REGION Network 96: Transfer P&P Left AxisX Home Interlock Condition
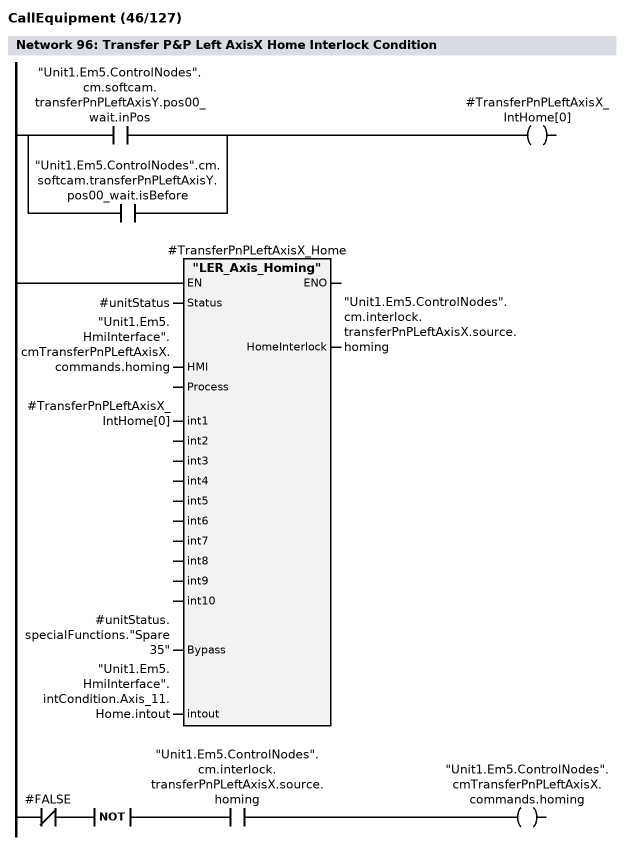
   RUNG wire#powerrail
      Contact( "Unit1.Em5.ControlNodes".cm.softcam.transferPnPLeftAxisY.pos00_wait.inPos )
      wire#w1
      Coil( #TransferPnPLeftAxisX_IntHome[0] )
   END_RUNG
   RUNG wire#powerrail
      Contact( "Unit1.Em5.ControlNodes".cm.softcam.transferPnPLeftAxisY.pos00_wait.isBefore )
   END_RUNG wire#w1
   RUNG wire#powerrail
      #TransferPnPLeftAxisX_Home(Status := #unitStatus, HMI := "Unit1.Em5.HmiInterface".cmTransferPnPLeftAxisX.commands.homing, Process :=, int1 := #TransferPnPLeftAxisX_IntHome[0], int2 :=, int3 :=, int4 :=, int5 :=, int6 :=, int7 :=, int8 :=, int9 :=, int10 :=, Bypass := #unitStatus.specialFunctions."Spare 35", intout := "Unit1.Em5.HmiInterface".intCondition.Axis_11.Home.intout, HomeInterlock => "Unit1.Em5.ControlNodes".cm.interlock.transferPnPLeftAxisX.source.homing)
   END_RUNG
   RUNG wire#powerrail
      I_Contact( #FALSE )
      Not()
      Contact( "Unit1.Em5.ControlNodes".cm.interlock.transferPnPLeftAxisX.source.homing )
      Coil( "Unit1.Em5.ControlNodes".cmTransferPnPLeftAxisX.commands.homing )
   END_RUNG
   // the same network as SCL:
   #TransferPnPLeftAxisX_IntHome[0] := "Unit1.Em5.ControlNodes".cm.softcam.transferPnPLeftAxisY.pos00_wait.inPos OR "Unit1.Em5.ControlNodes".cm.softcam.transferPnPLeftAxisY.pos00_wait.isBefore;
   #TransferPnPLeftAxisX_Home(Status := #unitStatus,   // "LER_Axis_Homing"
                           HMI := "Unit1.Em5.HmiInterface".cmTransferPnPLeftAxisX.commands.homing,
                           int1 := #TransferPnPLeftAxisX_IntHome[0],
                           Bypass := #unitStatus.specialFunctions."Spare 35",
                           intout := "Unit1.Em5.HmiInterface".intCondition.Axis_11.Home.intout,
                           HomeInterlock => "Unit1.Em5.ControlNodes".cm.interlock.transferPnPLeftAxisX.source.homing);
   "Unit1.Em5.ControlNodes".cmTransferPnPLeftAxisX.commands.homing := NOT (NOT #FALSE) AND "Unit1.Em5.ControlNodes".cm.interlock.transferPnPLeftAxisX.source.homing;
END_REGION

REGION Network 97: Transfer P&P Left AxisX JOG Interlock Condition
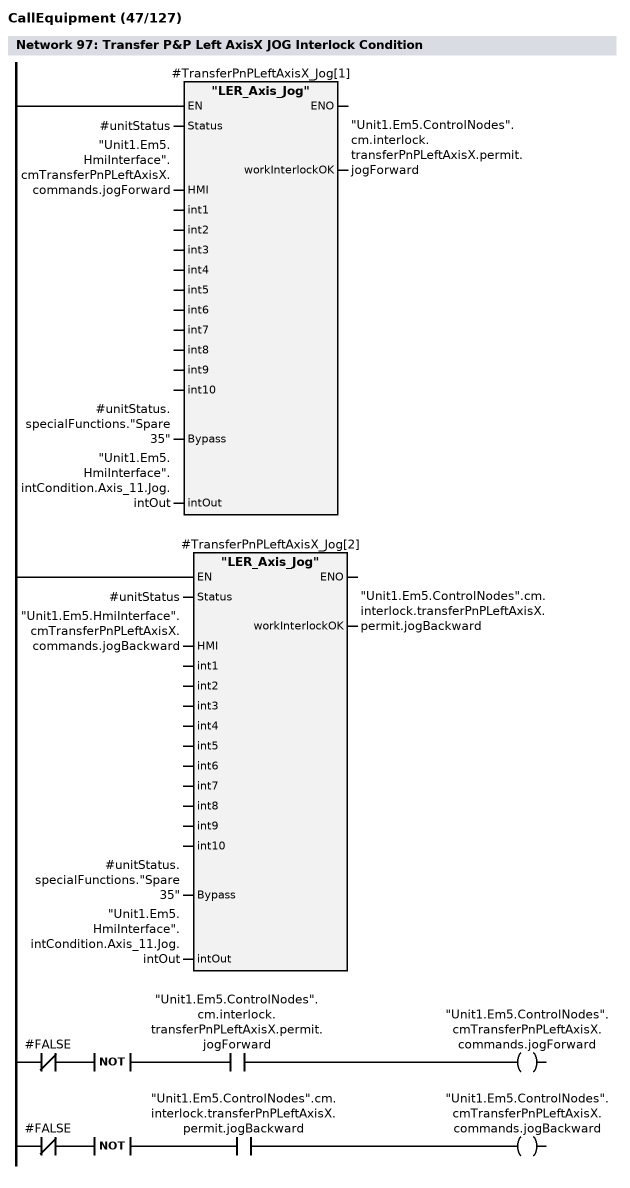
   RUNG wire#powerrail
      #TransferPnPLeftAxisX_Jog[1](Status := #unitStatus, HMI := "Unit1.Em5.HmiInterface".cmTransferPnPLeftAxisX.commands.jogForward, int1 :=, int2 :=, int3 :=, int4 :=, int5 :=, int6 :=, int7 :=, int8 :=, int9 :=, int10 :=, Bypass := #unitStatus.specialFunctions."Spare 35", intOut := "Unit1.Em5.HmiInterface".intCondition.Axis_11.Jog.intOut, workInterlockOK => "Unit1.Em5.ControlNodes".cm.interlock.transferPnPLeftAxisX.permit.jogForward)
   END_RUNG
   RUNG wire#powerrail
      #TransferPnPLeftAxisX_Jog[2](Status := #unitStatus, HMI := "Unit1.Em5.HmiInterface".cmTransferPnPLeftAxisX.commands.jogBackward, int1 :=, int2 :=, int3 :=, int4 :=, int5 :=, int6 :=, int7 :=, int8 :=, int9 :=, int10 :=, Bypass := #unitStatus.specialFunctions."Spare 35", intOut := "Unit1.Em5.HmiInterface".intCondition.Axis_11.Jog.intOut, workInterlockOK => "Unit1.Em5.ControlNodes".cm.interlock.transferPnPLeftAxisX.permit.jogBackward)
   END_RUNG
   RUNG wire#powerrail
      I_Contact( #FALSE )
      Not()
      Contact( "Unit1.Em5.ControlNodes".cm.interlock.transferPnPLeftAxisX.permit.jogForward )
      Coil( "Unit1.Em5.ControlNodes".cmTransferPnPLeftAxisX.commands.jogForward )
   END_RUNG
   RUNG wire#powerrail
      I_Contact( #FALSE )
      Not()
      Contact( "Unit1.Em5.ControlNodes".cm.interlock.transferPnPLeftAxisX.permit.jogBackward )
      Coil( "Unit1.Em5.ControlNodes".cmTransferPnPLeftAxisX.commands.jogBackward )
   END_RUNG
   // the same network as SCL:
   #TransferPnPLeftAxisX_Jog[1](Status := #unitStatus,   // "LER_Axis_Jog"
                           HMI := "Unit1.Em5.HmiInterface".cmTransferPnPLeftAxisX.commands.jogForward,
                           Bypass := #unitStatus.specialFunctions."Spare 35",
                           intOut := "Unit1.Em5.HmiInterface".intCondition.Axis_11.Jog.intOut,
                           workInterlockOK => "Unit1.Em5.ControlNodes".cm.interlock.transferPnPLeftAxisX.permit.jogForward);
   #TransferPnPLeftAxisX_Jog[2](Status := #unitStatus,   // "LER_Axis_Jog"
                           HMI := "Unit1.Em5.HmiInterface".cmTransferPnPLeftAxisX.commands.jogBackward,
                           Bypass := #unitStatus.specialFunctions."Spare 35",
                           intOut := "Unit1.Em5.HmiInterface".intCondition.Axis_11.Jog.intOut,
                           workInterlockOK => "Unit1.Em5.ControlNodes".cm.interlock.transferPnPLeftAxisX.permit.jogBackward);
   "Unit1.Em5.ControlNodes".cmTransferPnPLeftAxisX.commands.jogForward := NOT (NOT #FALSE) AND "Unit1.Em5.ControlNodes".cm.interlock.transferPnPLeftAxisX.permit.jogForward;
   "Unit1.Em5.ControlNodes".cmTransferPnPLeftAxisX.commands.jogBackward := NOT (NOT #FALSE) AND "Unit1.Em5.ControlNodes".cm.interlock.transferPnPLeftAxisX.permit.jogBackward;
END_REGION

REGION Network 98: Transfer P&P Left AxisX Position Absolute Position0
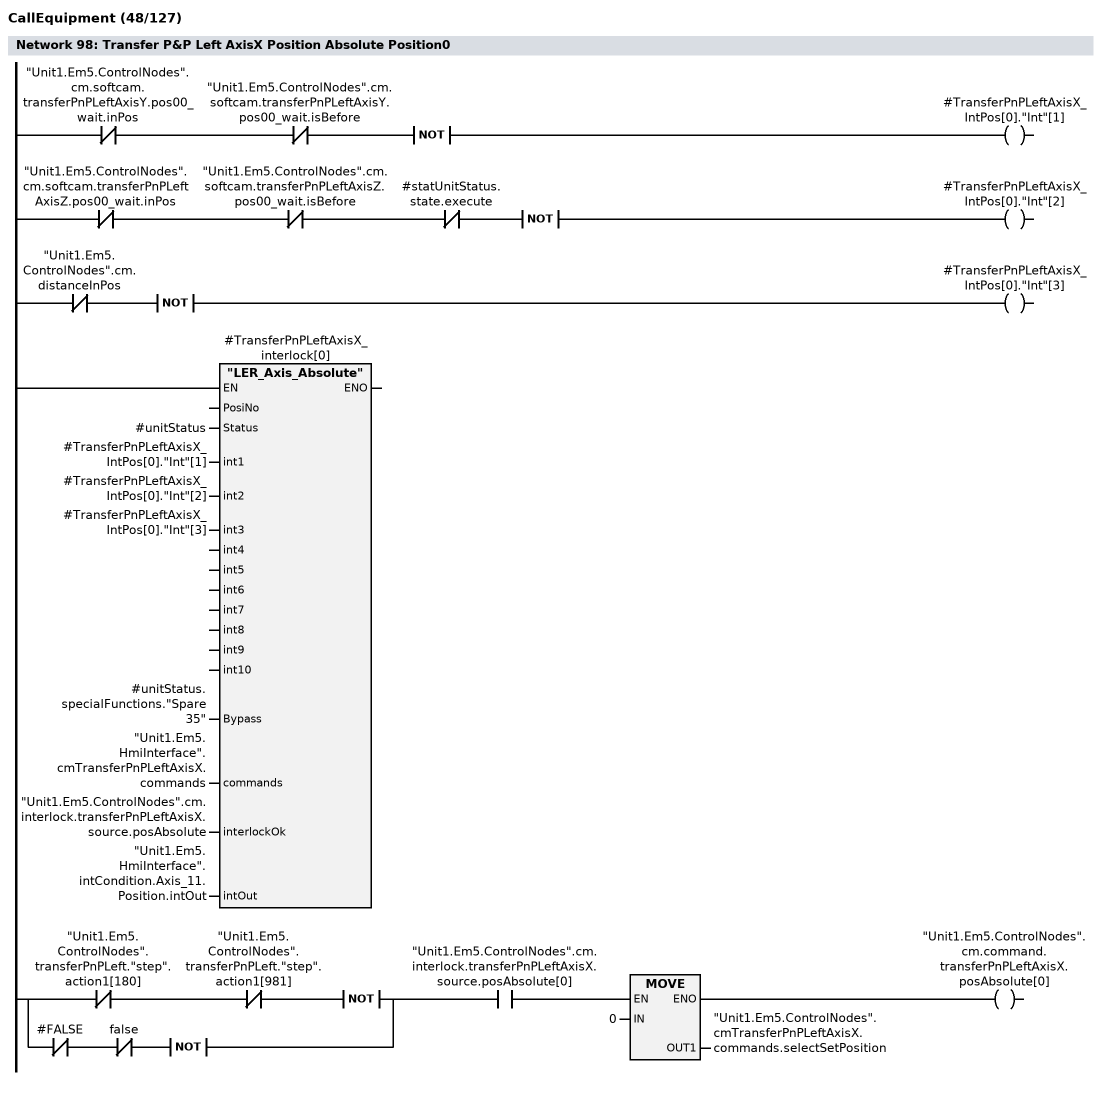
   RUNG wire#powerrail
      I_Contact( "Unit1.Em5.ControlNodes".cm.softcam.transferPnPLeftAxisY.pos00_wait.inPos )
      I_Contact( "Unit1.Em5.ControlNodes".cm.softcam.transferPnPLeftAxisY.pos00_wait.isBefore )
      Not()
      Coil( #TransferPnPLeftAxisX_IntPos[0]."Int"[1] )
   END_RUNG
   RUNG wire#powerrail
      I_Contact( "Unit1.Em5.ControlNodes".cm.softcam.transferPnPLeftAxisZ.pos00_wait.inPos )
      I_Contact( "Unit1.Em5.ControlNodes".cm.softcam.transferPnPLeftAxisZ.pos00_wait.isBefore )
      I_Contact( #statUnitStatus.state.execute )
      Not()
      Coil( #TransferPnPLeftAxisX_IntPos[0]."Int"[2] )
   END_RUNG
   RUNG wire#powerrail
      I_Contact( "Unit1.Em5.ControlNodes".cm.distanceInPos )
      Not()
      Coil( #TransferPnPLeftAxisX_IntPos[0]."Int"[3] )
   END_RUNG
   RUNG wire#powerrail
      #TransferPnPLeftAxisX_interlock[0](PosiNo :=, Status := #unitStatus, int1 := #TransferPnPLeftAxisX_IntPos[0]."Int"[1], int2 := #TransferPnPLeftAxisX_IntPos[0]."Int"[2], int3 := #TransferPnPLeftAxisX_IntPos[0]."Int"[3], int4 :=, int5 :=, int6 :=, int7 :=, int8 :=, int9 :=, int10 :=, Bypass := #unitStatus.specialFunctions."Spare 35", commands := "Unit1.Em5.HmiInterface".cmTransferPnPLeftAxisX.commands, interlockOk := "Unit1.Em5.ControlNodes".cm.interlock.transferPnPLeftAxisX.source.posAbsolute, intOut := "Unit1.Em5.HmiInterface".intCondition.Axis_11.Position.intOut)
   END_RUNG
   RUNG wire#powerrail
      I_Contact( "Unit1.Em5.ControlNodes".transferPnPLeft."step".action1[180] )
      I_Contact( "Unit1.Em5.ControlNodes".transferPnPLeft."step".action1[981] )
      Not()
      wire#w1
      Contact( "Unit1.Em5.ControlNodes".cm.interlock.transferPnPLeftAxisX.source.posAbsolute[0] )
      Move(in := 0, out1 => "Unit1.Em5.ControlNodes".cmTransferPnPLeftAxisX.commands.selectSetPosition)
      Coil( "Unit1.Em5.ControlNodes".cm.command.transferPnPLeftAxisX.posAbsolute[0] )
   END_RUNG
   RUNG wire#powerrail
      I_Contact( #FALSE )
      I_Contact( false )
      Not()
   END_RUNG wire#w1
   // the same network as SCL:
   #TransferPnPLeftAxisX_IntPos[0]."Int"[1] := NOT (NOT "Unit1.Em5.ControlNodes".cm.softcam.transferPnPLeftAxisY.pos00_wait.inPos AND NOT "Unit1.Em5.ControlNodes".cm.softcam.transferPnPLeftAxisY.pos00_wait.isBefore);
   #TransferPnPLeftAxisX_IntPos[0]."Int"[2] := NOT (NOT "Unit1.Em5.ControlNodes".cm.softcam.transferPnPLeftAxisZ.pos00_wait.inPos AND NOT "Unit1.Em5.ControlNodes".cm.softcam.transferPnPLeftAxisZ.pos00_wait.isBefore AND NOT #statUnitStatus.state.execute);
   #TransferPnPLeftAxisX_IntPos[0]."Int"[3] := NOT (NOT "Unit1.Em5.ControlNodes".cm.distanceInPos);
   #TransferPnPLeftAxisX_interlock[0](Status := #unitStatus,   // "LER_Axis_Absolute"
                           int1 := #TransferPnPLeftAxisX_IntPos[0]."Int"[1],
                           int2 := #TransferPnPLeftAxisX_IntPos[0]."Int"[2],
                           int3 := #TransferPnPLeftAxisX_IntPos[0]."Int"[3],
                           Bypass := #unitStatus.specialFunctions."Spare 35",
                           commands := "Unit1.Em5.HmiInterface".cmTransferPnPLeftAxisX.commands,
                           interlockOk := "Unit1.Em5.ControlNodes".cm.interlock.transferPnPLeftAxisX.source.posAbsolute,
                           intOut := "Unit1.Em5.HmiInterface".intCondition.Axis_11.Position.intOut);
   #_w1 := (NOT (NOT "Unit1.Em5.ControlNodes".transferPnPLeft."step".action1[180] AND NOT "Unit1.Em5.ControlNodes".transferPnPLeft."step".action1[981]) OR NOT (NOT #FALSE AND NOT false)) AND "Unit1.Em5.ControlNodes".cm.interlock.transferPnPLeftAxisX.source.posAbsolute[0];
   IF #_w1 THEN "Unit1.Em5.ControlNodes".cmTransferPnPLeftAxisX.commands.selectSetPosition := 0; END_IF;
   "Unit1.Em5.ControlNodes".cm.command.transferPnPLeftAxisX.posAbsolute[0] := #_w1;
END_REGION

REGION Network 99: Transfer P&P Left AxisX Position Absolute Position1
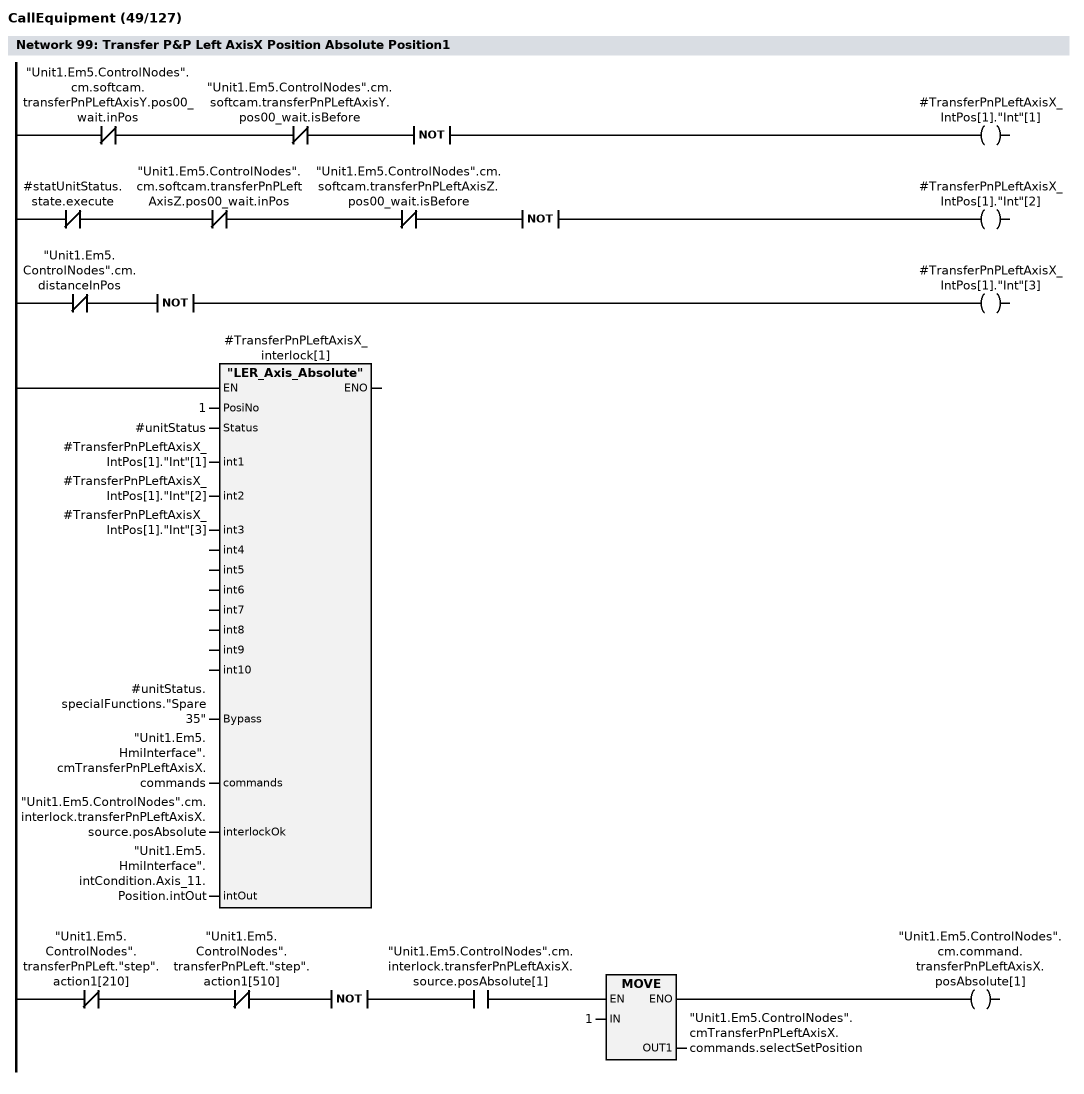
   RUNG wire#powerrail
      I_Contact( "Unit1.Em5.ControlNodes".cm.softcam.transferPnPLeftAxisY.pos00_wait.inPos )
      I_Contact( "Unit1.Em5.ControlNodes".cm.softcam.transferPnPLeftAxisY.pos00_wait.isBefore )
      Not()
      Coil( #TransferPnPLeftAxisX_IntPos[1]."Int"[1] )
   END_RUNG
   RUNG wire#powerrail
      I_Contact( #statUnitStatus.state.execute )
      I_Contact( "Unit1.Em5.ControlNodes".cm.softcam.transferPnPLeftAxisZ.pos00_wait.inPos )
      I_Contact( "Unit1.Em5.ControlNodes".cm.softcam.transferPnPLeftAxisZ.pos00_wait.isBefore )
      Not()
      Coil( #TransferPnPLeftAxisX_IntPos[1]."Int"[2] )
   END_RUNG
   RUNG wire#powerrail
      I_Contact( "Unit1.Em5.ControlNodes".cm.distanceInPos )
      Not()
      Coil( #TransferPnPLeftAxisX_IntPos[1]."Int"[3] )
   END_RUNG
   RUNG wire#powerrail
      #TransferPnPLeftAxisX_interlock[1](PosiNo := 1, Status := #unitStatus, int1 := #TransferPnPLeftAxisX_IntPos[1]."Int"[1], int2 := #TransferPnPLeftAxisX_IntPos[1]."Int"[2], int3 := #TransferPnPLeftAxisX_IntPos[1]."Int"[3], int4 :=, int5 :=, int6 :=, int7 :=, int8 :=, int9 :=, int10 :=, Bypass := #unitStatus.specialFunctions."Spare 35", commands := "Unit1.Em5.HmiInterface".cmTransferPnPLeftAxisX.commands, interlockOk := "Unit1.Em5.ControlNodes".cm.interlock.transferPnPLeftAxisX.source.posAbsolute, intOut := "Unit1.Em5.HmiInterface".intCondition.Axis_11.Position.intOut)
   END_RUNG
   RUNG wire#powerrail
      I_Contact( "Unit1.Em5.ControlNodes".transferPnPLeft."step".action1[210] )
      I_Contact( "Unit1.Em5.ControlNodes".transferPnPLeft."step".action1[510] )
      Not()
      Contact( "Unit1.Em5.ControlNodes".cm.interlock.transferPnPLeftAxisX.source.posAbsolute[1] )
      Move(in := 1, out1 => "Unit1.Em5.ControlNodes".cmTransferPnPLeftAxisX.commands.selectSetPosition)
      Coil( "Unit1.Em5.ControlNodes".cm.command.transferPnPLeftAxisX.posAbsolute[1] )
   END_RUNG
   // the same network as SCL:
   #TransferPnPLeftAxisX_IntPos[1]."Int"[1] := NOT (NOT "Unit1.Em5.ControlNodes".cm.softcam.transferPnPLeftAxisY.pos00_wait.inPos AND NOT "Unit1.Em5.ControlNodes".cm.softcam.transferPnPLeftAxisY.pos00_wait.isBefore);
   #TransferPnPLeftAxisX_IntPos[1]."Int"[2] := NOT (NOT #statUnitStatus.state.execute AND NOT "Unit1.Em5.ControlNodes".cm.softcam.transferPnPLeftAxisZ.pos00_wait.inPos AND NOT "Unit1.Em5.ControlNodes".cm.softcam.transferPnPLeftAxisZ.pos00_wait.isBefore);
   #TransferPnPLeftAxisX_IntPos[1]."Int"[3] := NOT (NOT "Unit1.Em5.ControlNodes".cm.distanceInPos);
   #TransferPnPLeftAxisX_interlock[1](PosiNo := 1,   // "LER_Axis_Absolute"
                           Status := #unitStatus,
                           int1 := #TransferPnPLeftAxisX_IntPos[1]."Int"[1],
                           int2 := #TransferPnPLeftAxisX_IntPos[1]."Int"[2],
                           int3 := #TransferPnPLeftAxisX_IntPos[1]."Int"[3],
                           Bypass := #unitStatus.specialFunctions."Spare 35",
                           commands := "Unit1.Em5.HmiInterface".cmTransferPnPLeftAxisX.commands,
                           interlockOk := "Unit1.Em5.ControlNodes".cm.interlock.transferPnPLeftAxisX.source.posAbsolute,
                           intOut := "Unit1.Em5.HmiInterface".intCondition.Axis_11.Position.intOut);
   #_w1 := NOT (NOT "Unit1.Em5.ControlNodes".transferPnPLeft."step".action1[210] AND NOT "Unit1.Em5.ControlNodes".transferPnPLeft."step".action1[510]) AND "Unit1.Em5.ControlNodes".cm.interlock.transferPnPLeftAxisX.source.posAbsolute[1];
   IF #_w1 THEN "Unit1.Em5.ControlNodes".cmTransferPnPLeftAxisX.commands.selectSetPosition := 1; END_IF;
   "Unit1.Em5.ControlNodes".cm.command.transferPnPLeftAxisX.posAbsolute[1] := #_w1;
END_REGION

REGION Network 100: Transfer P&P Left AxisX Position Absolute Position2
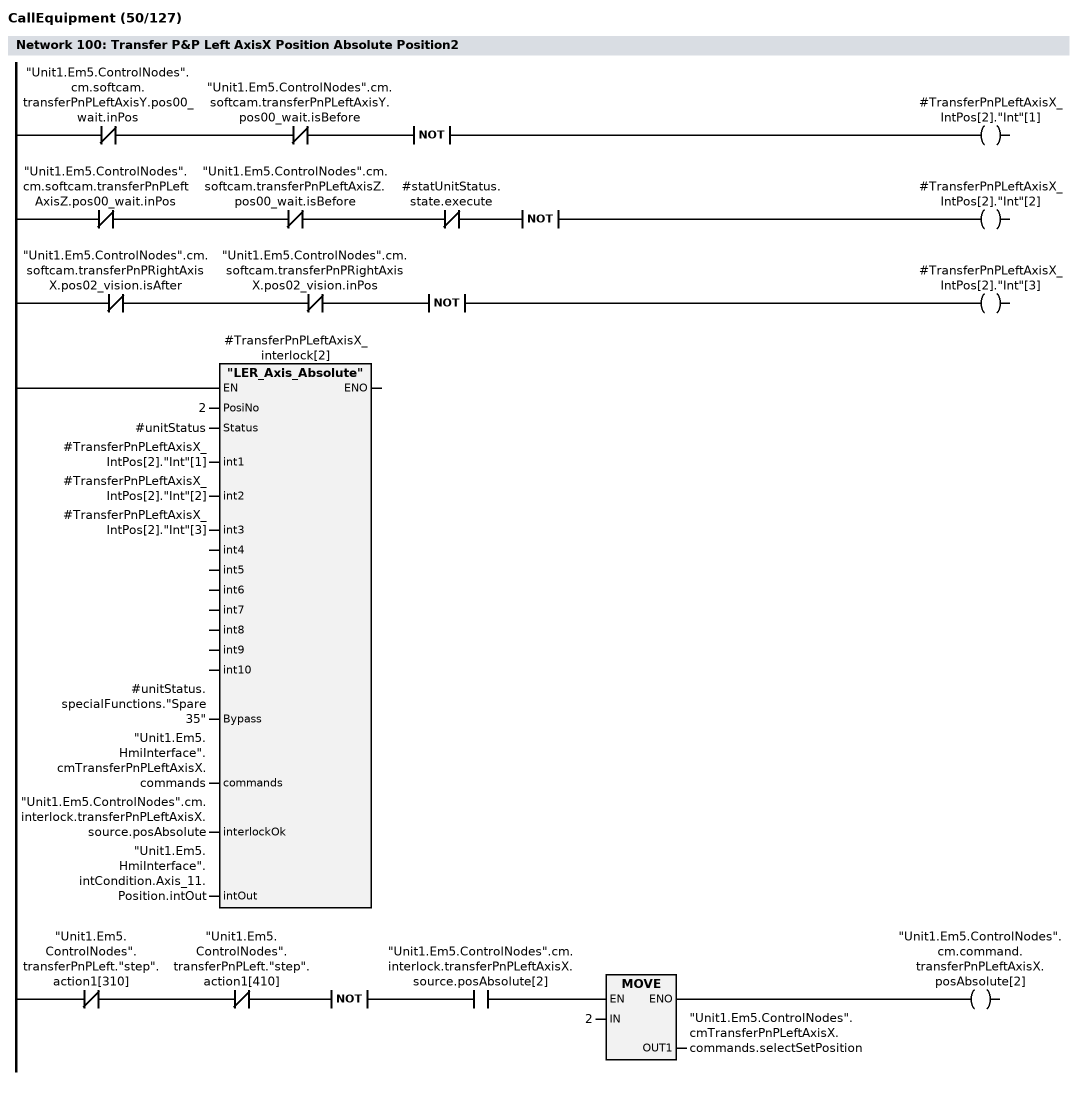
   RUNG wire#powerrail
      I_Contact( "Unit1.Em5.ControlNodes".cm.softcam.transferPnPLeftAxisY.pos00_wait.inPos )
      I_Contact( "Unit1.Em5.ControlNodes".cm.softcam.transferPnPLeftAxisY.pos00_wait.isBefore )
      Not()
      Coil( #TransferPnPLeftAxisX_IntPos[2]."Int"[1] )
   END_RUNG
   RUNG wire#powerrail
      I_Contact( "Unit1.Em5.ControlNodes".cm.softcam.transferPnPLeftAxisZ.pos00_wait.inPos )
      I_Contact( "Unit1.Em5.ControlNodes".cm.softcam.transferPnPLeftAxisZ.pos00_wait.isBefore )
      I_Contact( #statUnitStatus.state.execute )
      Not()
      Coil( #TransferPnPLeftAxisX_IntPos[2]."Int"[2] )
   END_RUNG
   RUNG wire#powerrail
      I_Contact( "Unit1.Em5.ControlNodes".cm.softcam.transferPnPRightAxisX.pos02_vision.isAfter )
      I_Contact( "Unit1.Em5.ControlNodes".cm.softcam.transferPnPRightAxisX.pos02_vision.inPos )
      Not()
      Coil( #TransferPnPLeftAxisX_IntPos[2]."Int"[3] )
   END_RUNG
   RUNG wire#powerrail
      #TransferPnPLeftAxisX_interlock[2](PosiNo := 2, Status := #unitStatus, int1 := #TransferPnPLeftAxisX_IntPos[2]."Int"[1], int2 := #TransferPnPLeftAxisX_IntPos[2]."Int"[2], int3 := #TransferPnPLeftAxisX_IntPos[2]."Int"[3], int4 :=, int5 :=, int6 :=, int7 :=, int8 :=, int9 :=, int10 :=, Bypass := #unitStatus.specialFunctions."Spare 35", commands := "Unit1.Em5.HmiInterface".cmTransferPnPLeftAxisX.commands, interlockOk := "Unit1.Em5.ControlNodes".cm.interlock.transferPnPLeftAxisX.source.posAbsolute, intOut := "Unit1.Em5.HmiInterface".intCondition.Axis_11.Position.intOut)
   END_RUNG
   RUNG wire#powerrail
      I_Contact( "Unit1.Em5.ControlNodes".transferPnPLeft."step".action1[310] )
      I_Contact( "Unit1.Em5.ControlNodes".transferPnPLeft."step".action1[410] )
      Not()
      Contact( "Unit1.Em5.ControlNodes".cm.interlock.transferPnPLeftAxisX.source.posAbsolute[2] )
      Move(in := 2, out1 => "Unit1.Em5.ControlNodes".cmTransferPnPLeftAxisX.commands.selectSetPosition)
      Coil( "Unit1.Em5.ControlNodes".cm.command.transferPnPLeftAxisX.posAbsolute[2] )
   END_RUNG
   // the same network as SCL:
   #TransferPnPLeftAxisX_IntPos[2]."Int"[1] := NOT (NOT "Unit1.Em5.ControlNodes".cm.softcam.transferPnPLeftAxisY.pos00_wait.inPos AND NOT "Unit1.Em5.ControlNodes".cm.softcam.transferPnPLeftAxisY.pos00_wait.isBefore);
   #TransferPnPLeftAxisX_IntPos[2]."Int"[2] := NOT (NOT "Unit1.Em5.ControlNodes".cm.softcam.transferPnPLeftAxisZ.pos00_wait.inPos AND NOT "Unit1.Em5.ControlNodes".cm.softcam.transferPnPLeftAxisZ.pos00_wait.isBefore AND NOT #statUnitStatus.state.execute);
   #TransferPnPLeftAxisX_IntPos[2]."Int"[3] := NOT (NOT "Unit1.Em5.ControlNodes".cm.softcam.transferPnPRightAxisX.pos02_vision.isAfter AND NOT "Unit1.Em5.ControlNodes".cm.softcam.transferPnPRightAxisX.pos02_vision.inPos);
   #TransferPnPLeftAxisX_interlock[2](PosiNo := 2,   // "LER_Axis_Absolute"
                           Status := #unitStatus,
                           int1 := #TransferPnPLeftAxisX_IntPos[2]."Int"[1],
                           int2 := #TransferPnPLeftAxisX_IntPos[2]."Int"[2],
                           int3 := #TransferPnPLeftAxisX_IntPos[2]."Int"[3],
                           Bypass := #unitStatus.specialFunctions."Spare 35",
                           commands := "Unit1.Em5.HmiInterface".cmTransferPnPLeftAxisX.commands,
                           interlockOk := "Unit1.Em5.ControlNodes".cm.interlock.transferPnPLeftAxisX.source.posAbsolute,
                           intOut := "Unit1.Em5.HmiInterface".intCondition.Axis_11.Position.intOut);
   #_w1 := NOT (NOT "Unit1.Em5.ControlNodes".transferPnPLeft."step".action1[310] AND NOT "Unit1.Em5.ControlNodes".transferPnPLeft."step".action1[410]) AND "Unit1.Em5.ControlNodes".cm.interlock.transferPnPLeftAxisX.source.posAbsolute[2];
   IF #_w1 THEN "Unit1.Em5.ControlNodes".cmTransferPnPLeftAxisX.commands.selectSetPosition := 2; END_IF;
   "Unit1.Em5.ControlNodes".cm.command.transferPnPLeftAxisX.posAbsolute[2] := #_w1;
END_REGION

REGION Network 101: Transfer P&P Left AxisX Position Absolute Position3
   // Jump : sequence doublecheck position with tr right pp
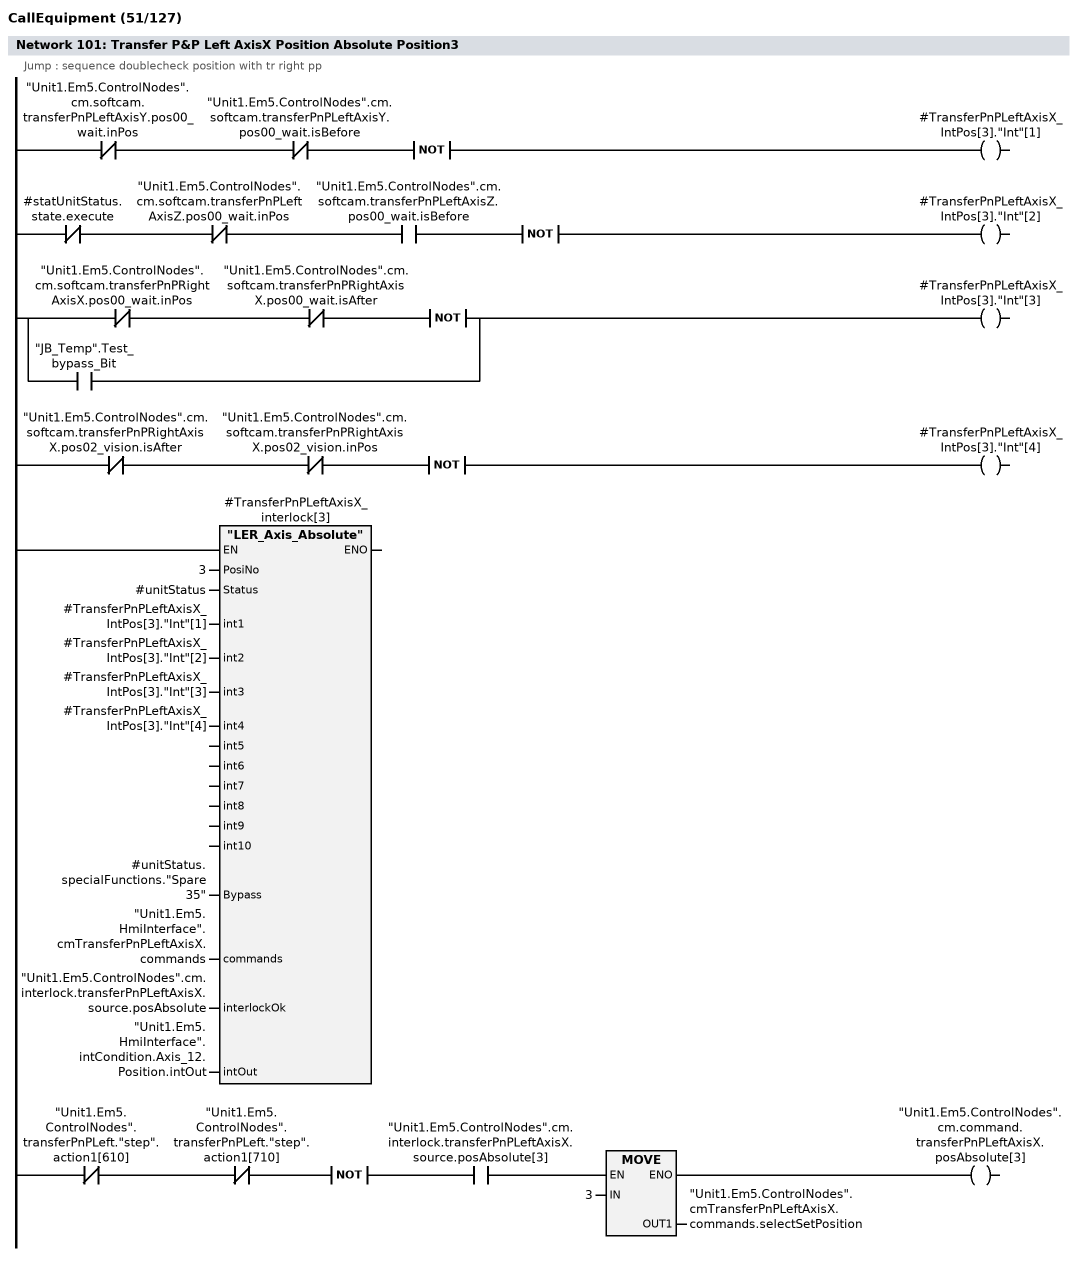
   RUNG wire#powerrail
      I_Contact( "Unit1.Em5.ControlNodes".cm.softcam.transferPnPLeftAxisY.pos00_wait.inPos )
      I_Contact( "Unit1.Em5.ControlNodes".cm.softcam.transferPnPLeftAxisY.pos00_wait.isBefore )
      Not()
      Coil( #TransferPnPLeftAxisX_IntPos[3]."Int"[1] )
   END_RUNG
   RUNG wire#powerrail
      I_Contact( #statUnitStatus.state.execute )
      I_Contact( "Unit1.Em5.ControlNodes".cm.softcam.transferPnPLeftAxisZ.pos00_wait.inPos )
      Contact( "Unit1.Em5.ControlNodes".cm.softcam.transferPnPLeftAxisZ.pos00_wait.isBefore )
      Not()
      Coil( #TransferPnPLeftAxisX_IntPos[3]."Int"[2] )
   END_RUNG
   RUNG wire#powerrail
      I_Contact( "Unit1.Em5.ControlNodes".cm.softcam.transferPnPRightAxisX.pos00_wait.inPos )
      I_Contact( "Unit1.Em5.ControlNodes".cm.softcam.transferPnPRightAxisX.pos00_wait.isAfter )
      Not()
      wire#w1
      Coil( #TransferPnPLeftAxisX_IntPos[3]."Int"[3] )
   END_RUNG
   RUNG wire#powerrail
      Contact( "JB_Temp".Test_bypass_Bit )
   END_RUNG wire#w1
   RUNG wire#powerrail
      I_Contact( "Unit1.Em5.ControlNodes".cm.softcam.transferPnPRightAxisX.pos02_vision.isAfter )
      I_Contact( "Unit1.Em5.ControlNodes".cm.softcam.transferPnPRightAxisX.pos02_vision.inPos )
      Not()
      Coil( #TransferPnPLeftAxisX_IntPos[3]."Int"[4] )
   END_RUNG
   RUNG wire#powerrail
      #TransferPnPLeftAxisX_interlock[3](PosiNo := 3, Status := #unitStatus, int1 := #TransferPnPLeftAxisX_IntPos[3]."Int"[1], int2 := #TransferPnPLeftAxisX_IntPos[3]."Int"[2], int3 := #TransferPnPLeftAxisX_IntPos[3]."Int"[3], int4 := #TransferPnPLeftAxisX_IntPos[3]."Int"[4], int5 :=, int6 :=, int7 :=, int8 :=, int9 :=, int10 :=, Bypass := #unitStatus.specialFunctions."Spare 35", commands := "Unit1.Em5.HmiInterface".cmTransferPnPLeftAxisX.commands, interlockOk := "Unit1.Em5.ControlNodes".cm.interlock.transferPnPLeftAxisX.source.posAbsolute, intOut := "Unit1.Em5.HmiInterface".intCondition.Axis_12.Position.intOut)
   END_RUNG
   RUNG wire#powerrail
      I_Contact( "Unit1.Em5.ControlNodes".transferPnPLeft."step".action1[610] )
      I_Contact( "Unit1.Em5.ControlNodes".transferPnPLeft."step".action1[710] )
      Not()
      Contact( "Unit1.Em5.ControlNodes".cm.interlock.transferPnPLeftAxisX.source.posAbsolute[3] )
      Move(in := 3, out1 => "Unit1.Em5.ControlNodes".cmTransferPnPLeftAxisX.commands.selectSetPosition)
      Coil( "Unit1.Em5.ControlNodes".cm.command.transferPnPLeftAxisX.posAbsolute[3] )
   END_RUNG
   // the same network as SCL:
   #TransferPnPLeftAxisX_IntPos[3]."Int"[1] := NOT (NOT "Unit1.Em5.ControlNodes".cm.softcam.transferPnPLeftAxisY.pos00_wait.inPos AND NOT "Unit1.Em5.ControlNodes".cm.softcam.transferPnPLeftAxisY.pos00_wait.isBefore);
   #TransferPnPLeftAxisX_IntPos[3]."Int"[2] := NOT (NOT #statUnitStatus.state.execute AND NOT "Unit1.Em5.ControlNodes".cm.softcam.transferPnPLeftAxisZ.pos00_wait.inPos AND "Unit1.Em5.ControlNodes".cm.softcam.transferPnPLeftAxisZ.pos00_wait.isBefore);
   #TransferPnPLeftAxisX_IntPos[3]."Int"[3] := NOT (NOT "Unit1.Em5.ControlNodes".cm.softcam.transferPnPRightAxisX.pos00_wait.inPos AND NOT "Unit1.Em5.ControlNodes".cm.softcam.transferPnPRightAxisX.pos00_wait.isAfter) OR "JB_Temp".Test_bypass_Bit;
   #TransferPnPLeftAxisX_IntPos[3]."Int"[4] := NOT (NOT "Unit1.Em5.ControlNodes".cm.softcam.transferPnPRightAxisX.pos02_vision.isAfter AND NOT "Unit1.Em5.ControlNodes".cm.softcam.transferPnPRightAxisX.pos02_vision.inPos);
   #TransferPnPLeftAxisX_interlock[3](PosiNo := 3,   // "LER_Axis_Absolute"
                           Status := #unitStatus,
                           int1 := #TransferPnPLeftAxisX_IntPos[3]."Int"[1],
                           int2 := #TransferPnPLeftAxisX_IntPos[3]."Int"[2],
                           int3 := #TransferPnPLeftAxisX_IntPos[3]."Int"[3],
                           int4 := #TransferPnPLeftAxisX_IntPos[3]."Int"[4],
                           Bypass := #unitStatus.specialFunctions."Spare 35",
                           commands := "Unit1.Em5.HmiInterface".cmTransferPnPLeftAxisX.commands,
                           interlockOk := "Unit1.Em5.ControlNodes".cm.interlock.transferPnPLeftAxisX.source.posAbsolute,
                           intOut := "Unit1.Em5.HmiInterface".intCondition.Axis_12.Position.intOut);
   #_w1 := NOT (NOT "Unit1.Em5.ControlNodes".transferPnPLeft."step".action1[610] AND NOT "Unit1.Em5.ControlNodes".transferPnPLeft."step".action1[710]) AND "Unit1.Em5.ControlNodes".cm.interlock.transferPnPLeftAxisX.source.posAbsolute[3];
   IF #_w1 THEN "Unit1.Em5.ControlNodes".cmTransferPnPLeftAxisX.commands.selectSetPosition := 3; END_IF;
   "Unit1.Em5.ControlNodes".cm.command.transferPnPLeftAxisX.posAbsolute[3] := #_w1;
END_REGION

REGION Network 102: Transfer P&P Left AxisX Position Absolute Position4
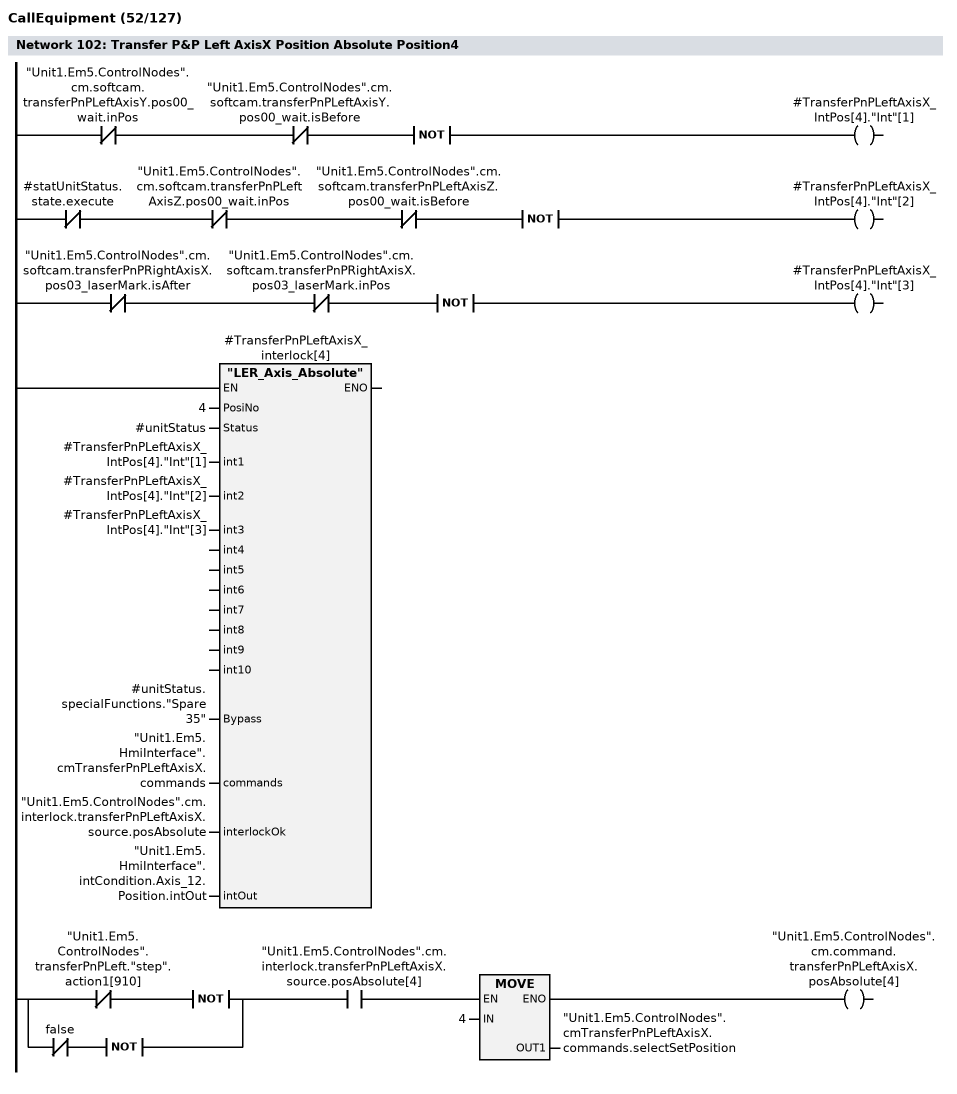
   RUNG wire#powerrail
      I_Contact( "Unit1.Em5.ControlNodes".cm.softcam.transferPnPLeftAxisY.pos00_wait.inPos )
      I_Contact( "Unit1.Em5.ControlNodes".cm.softcam.transferPnPLeftAxisY.pos00_wait.isBefore )
      Not()
      Coil( #TransferPnPLeftAxisX_IntPos[4]."Int"[1] )
   END_RUNG
   RUNG wire#powerrail
      I_Contact( #statUnitStatus.state.execute )
      I_Contact( "Unit1.Em5.ControlNodes".cm.softcam.transferPnPLeftAxisZ.pos00_wait.inPos )
      I_Contact( "Unit1.Em5.ControlNodes".cm.softcam.transferPnPLeftAxisZ.pos00_wait.isBefore )
      Not()
      Coil( #TransferPnPLeftAxisX_IntPos[4]."Int"[2] )
   END_RUNG
   RUNG wire#powerrail
      I_Contact( "Unit1.Em5.ControlNodes".cm.softcam.transferPnPRightAxisX.pos03_laserMark.isAfter )
      I_Contact( "Unit1.Em5.ControlNodes".cm.softcam.transferPnPRightAxisX.pos03_laserMark.inPos )
      Not()
      Coil( #TransferPnPLeftAxisX_IntPos[4]."Int"[3] )
   END_RUNG
   RUNG wire#powerrail
      #TransferPnPLeftAxisX_interlock[4](PosiNo := 4, Status := #unitStatus, int1 := #TransferPnPLeftAxisX_IntPos[4]."Int"[1], int2 := #TransferPnPLeftAxisX_IntPos[4]."Int"[2], int3 := #TransferPnPLeftAxisX_IntPos[4]."Int"[3], int4 :=, int5 :=, int6 :=, int7 :=, int8 :=, int9 :=, int10 :=, Bypass := #unitStatus.specialFunctions."Spare 35", commands := "Unit1.Em5.HmiInterface".cmTransferPnPLeftAxisX.commands, interlockOk := "Unit1.Em5.ControlNodes".cm.interlock.transferPnPLeftAxisX.source.posAbsolute, intOut := "Unit1.Em5.HmiInterface".intCondition.Axis_12.Position.intOut)
   END_RUNG
   RUNG wire#powerrail
      I_Contact( "Unit1.Em5.ControlNodes".transferPnPLeft."step".action1[910] )
      Not()
      wire#w1
      Contact( "Unit1.Em5.ControlNodes".cm.interlock.transferPnPLeftAxisX.source.posAbsolute[4] )
      Move(in := 4, out1 => "Unit1.Em5.ControlNodes".cmTransferPnPLeftAxisX.commands.selectSetPosition)
      Coil( "Unit1.Em5.ControlNodes".cm.command.transferPnPLeftAxisX.posAbsolute[4] )
   END_RUNG
   RUNG wire#powerrail
      I_Contact( false )
      Not()
   END_RUNG wire#w1
   // the same network as SCL:
   #TransferPnPLeftAxisX_IntPos[4]."Int"[1] := NOT (NOT "Unit1.Em5.ControlNodes".cm.softcam.transferPnPLeftAxisY.pos00_wait.inPos AND NOT "Unit1.Em5.ControlNodes".cm.softcam.transferPnPLeftAxisY.pos00_wait.isBefore);
   #TransferPnPLeftAxisX_IntPos[4]."Int"[2] := NOT (NOT #statUnitStatus.state.execute AND NOT "Unit1.Em5.ControlNodes".cm.softcam.transferPnPLeftAxisZ.pos00_wait.inPos AND NOT "Unit1.Em5.ControlNodes".cm.softcam.transferPnPLeftAxisZ.pos00_wait.isBefore);
   #TransferPnPLeftAxisX_IntPos[4]."Int"[3] := NOT (NOT "Unit1.Em5.ControlNodes".cm.softcam.transferPnPRightAxisX.pos03_laserMark.isAfter AND NOT "Unit1.Em5.ControlNodes".cm.softcam.transferPnPRightAxisX.pos03_laserMark.inPos);
   #TransferPnPLeftAxisX_interlock[4](PosiNo := 4,   // "LER_Axis_Absolute"
                           Status := #unitStatus,
                           int1 := #TransferPnPLeftAxisX_IntPos[4]."Int"[1],
                           int2 := #TransferPnPLeftAxisX_IntPos[4]."Int"[2],
                           int3 := #TransferPnPLeftAxisX_IntPos[4]."Int"[3],
                           Bypass := #unitStatus.specialFunctions."Spare 35",
                           commands := "Unit1.Em5.HmiInterface".cmTransferPnPLeftAxisX.commands,
                           interlockOk := "Unit1.Em5.ControlNodes".cm.interlock.transferPnPLeftAxisX.source.posAbsolute,
                           intOut := "Unit1.Em5.HmiInterface".intCondition.Axis_12.Position.intOut);
   #_w1 := (NOT (NOT "Unit1.Em5.ControlNodes".transferPnPLeft."step".action1[910]) OR NOT (NOT false)) AND "Unit1.Em5.ControlNodes".cm.interlock.transferPnPLeftAxisX.source.posAbsolute[4];
   IF #_w1 THEN "Unit1.Em5.ControlNodes".cmTransferPnPLeftAxisX.commands.selectSetPosition := 4; END_IF;
   "Unit1.Em5.ControlNodes".cm.command.transferPnPLeftAxisX.posAbsolute[4] := #_w1;
END_REGION

REGION Network 103: Transfer P&P Left AxisX Position Absolute Position5
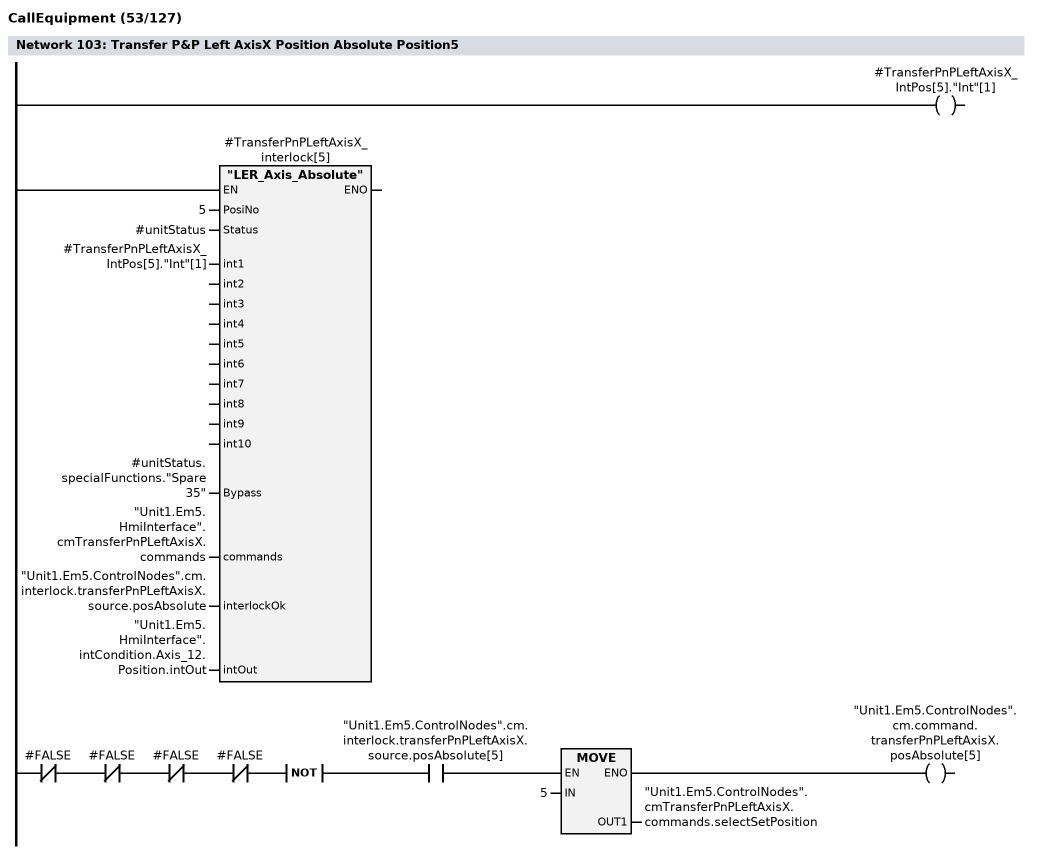
   RUNG wire#powerrail
      Coil( #TransferPnPLeftAxisX_IntPos[5]."Int"[1] )
   END_RUNG
   RUNG wire#powerrail
      #TransferPnPLeftAxisX_interlock[5](PosiNo := 5, Status := #unitStatus, int1 := #TransferPnPLeftAxisX_IntPos[5]."Int"[1], int2 :=, int3 :=, int4 :=, int5 :=, int6 :=, int7 :=, int8 :=, int9 :=, int10 :=, Bypass := #unitStatus.specialFunctions."Spare 35", commands := "Unit1.Em5.HmiInterface".cmTransferPnPLeftAxisX.commands, interlockOk := "Unit1.Em5.ControlNodes".cm.interlock.transferPnPLeftAxisX.source.posAbsolute, intOut := "Unit1.Em5.HmiInterface".intCondition.Axis_12.Position.intOut)
   END_RUNG
   RUNG wire#powerrail
      I_Contact( #FALSE )
      I_Contact( #FALSE )
      I_Contact( #FALSE )
      I_Contact( #FALSE )
      Not()
      Contact( "Unit1.Em5.ControlNodes".cm.interlock.transferPnPLeftAxisX.source.posAbsolute[5] )
      Move(in := 5, out1 => "Unit1.Em5.ControlNodes".cmTransferPnPLeftAxisX.commands.selectSetPosition)
      Coil( "Unit1.Em5.ControlNodes".cm.command.transferPnPLeftAxisX.posAbsolute[5] )
   END_RUNG
   // the same network as SCL:
   #TransferPnPLeftAxisX_IntPos[5]."Int"[1] := TRUE;
   #TransferPnPLeftAxisX_interlock[5](PosiNo := 5,   // "LER_Axis_Absolute"
                           Status := #unitStatus,
                           int1 := #TransferPnPLeftAxisX_IntPos[5]."Int"[1],
                           Bypass := #unitStatus.specialFunctions."Spare 35",
                           commands := "Unit1.Em5.HmiInterface".cmTransferPnPLeftAxisX.commands,
                           interlockOk := "Unit1.Em5.ControlNodes".cm.interlock.transferPnPLeftAxisX.source.posAbsolute,
                           intOut := "Unit1.Em5.HmiInterface".intCondition.Axis_12.Position.intOut);
   #_w1 := NOT (NOT #FALSE AND NOT #FALSE AND NOT #FALSE AND NOT #FALSE) AND "Unit1.Em5.ControlNodes".cm.interlock.transferPnPLeftAxisX.source.posAbsolute[5];
   IF #_w1 THEN "Unit1.Em5.ControlNodes".cmTransferPnPLeftAxisX.commands.selectSetPosition := 5; END_IF;
   "Unit1.Em5.ControlNodes".cm.command.transferPnPLeftAxisX.posAbsolute[5] := #_w1;
END_REGION

REGION Network 104: Transfer P&P Left AxisX Position Absolute Position7
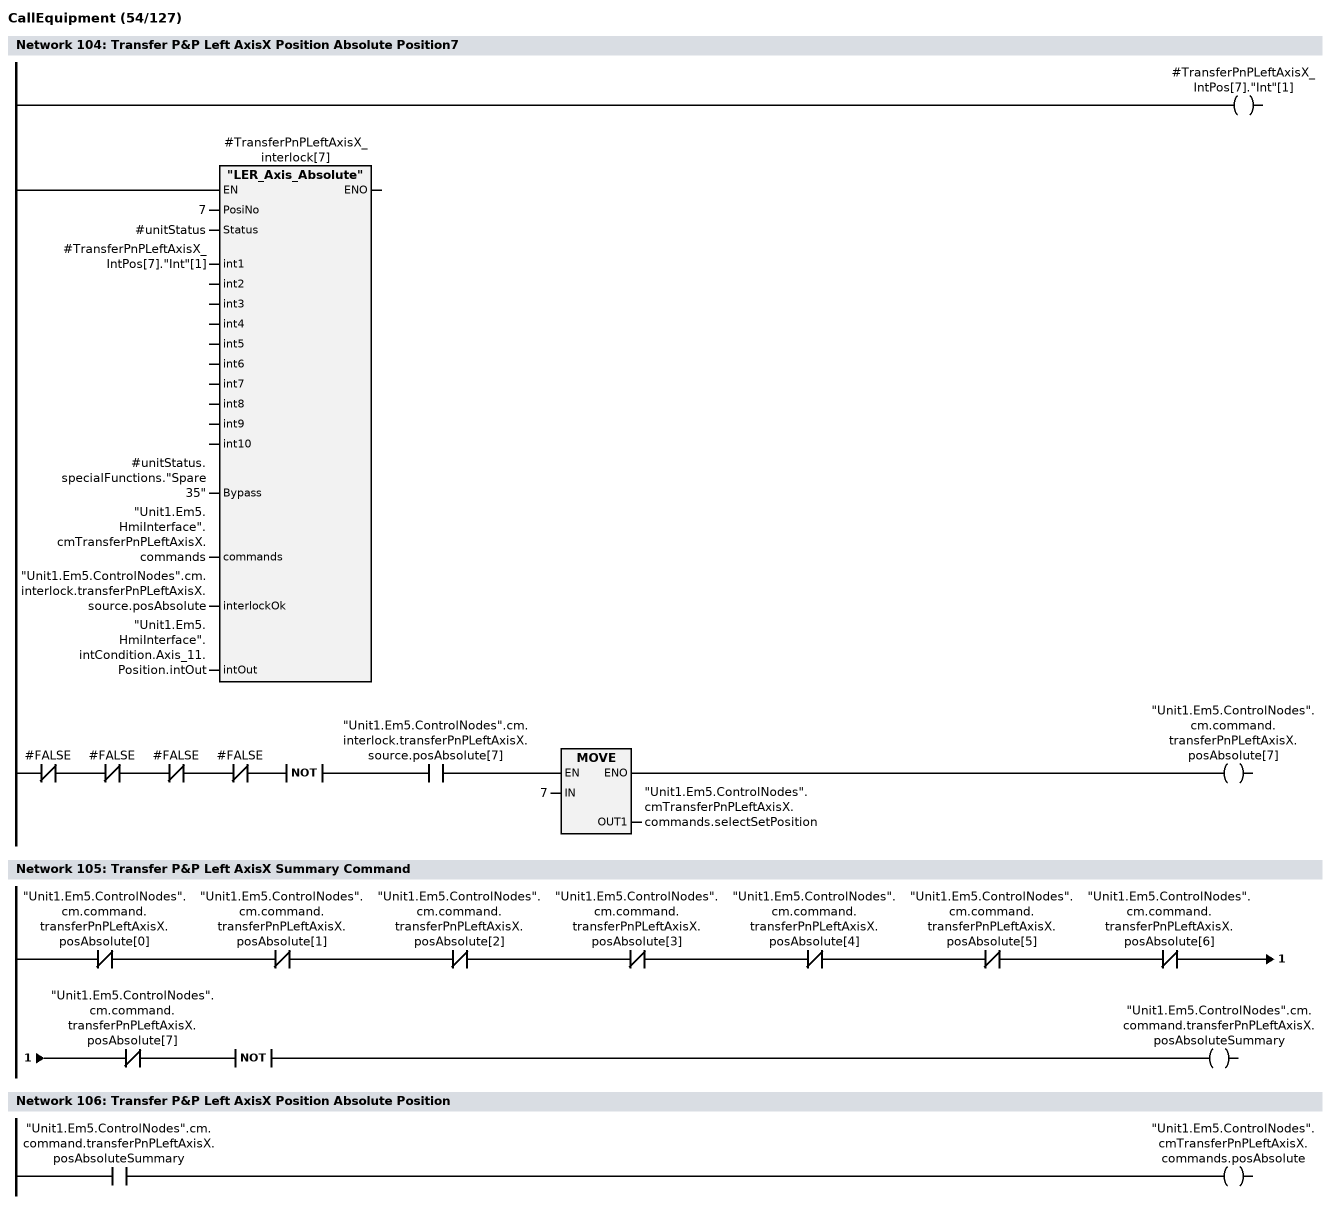
   RUNG wire#powerrail
      Coil( #TransferPnPLeftAxisX_IntPos[7]."Int"[1] )
   END_RUNG
   RUNG wire#powerrail
      #TransferPnPLeftAxisX_interlock[7](PosiNo := 7, Status := #unitStatus, int1 := #TransferPnPLeftAxisX_IntPos[7]."Int"[1], int2 :=, int3 :=, int4 :=, int5 :=, int6 :=, int7 :=, int8 :=, int9 :=, int10 :=, Bypass := #unitStatus.specialFunctions."Spare 35", commands := "Unit1.Em5.HmiInterface".cmTransferPnPLeftAxisX.commands, interlockOk := "Unit1.Em5.ControlNodes".cm.interlock.transferPnPLeftAxisX.source.posAbsolute, intOut := "Unit1.Em5.HmiInterface".intCondition.Axis_11.Position.intOut)
   END_RUNG
   RUNG wire#powerrail
      I_Contact( #FALSE )
      I_Contact( #FALSE )
      I_Contact( #FALSE )
      I_Contact( #FALSE )
      Not()
      Contact( "Unit1.Em5.ControlNodes".cm.interlock.transferPnPLeftAxisX.source.posAbsolute[7] )
      Move(in := 7, out1 => "Unit1.Em5.ControlNodes".cmTransferPnPLeftAxisX.commands.selectSetPosition)
      Coil( "Unit1.Em5.ControlNodes".cm.command.transferPnPLeftAxisX.posAbsolute[7] )
   END_RUNG
   // the same network as SCL:
   #TransferPnPLeftAxisX_IntPos[7]."Int"[1] := TRUE;
   #TransferPnPLeftAxisX_interlock[7](PosiNo := 7,   // "LER_Axis_Absolute"
                           Status := #unitStatus,
                           int1 := #TransferPnPLeftAxisX_IntPos[7]."Int"[1],
                           Bypass := #unitStatus.specialFunctions."Spare 35",
                           commands := "Unit1.Em5.HmiInterface".cmTransferPnPLeftAxisX.commands,
                           interlockOk := "Unit1.Em5.ControlNodes".cm.interlock.transferPnPLeftAxisX.source.posAbsolute,
                           intOut := "Unit1.Em5.HmiInterface".intCondition.Axis_11.Position.intOut);
   #_w1 := NOT (NOT #FALSE AND NOT #FALSE AND NOT #FALSE AND NOT #FALSE) AND "Unit1.Em5.ControlNodes".cm.interlock.transferPnPLeftAxisX.source.posAbsolute[7];
   IF #_w1 THEN "Unit1.Em5.ControlNodes".cmTransferPnPLeftAxisX.commands.selectSetPosition := 7; END_IF;
   "Unit1.Em5.ControlNodes".cm.command.transferPnPLeftAxisX.posAbsolute[7] := #_w1;
END_REGION

REGION Network 105: Transfer P&P Left AxisX Summary Command
   RUNG wire#powerrail
      I_Contact( "Unit1.Em5.ControlNodes".cm.command.transferPnPLeftAxisX.posAbsolute[0] )
      I_Contact( "Unit1.Em5.ControlNodes".cm.command.transferPnPLeftAxisX.posAbsolute[1] )
      I_Contact( "Unit1.Em5.ControlNodes".cm.command.transferPnPLeftAxisX.posAbsolute[2] )
      I_Contact( "Unit1.Em5.ControlNodes".cm.command.transferPnPLeftAxisX.posAbsolute[3] )
      I_Contact( "Unit1.Em5.ControlNodes".cm.command.transferPnPLeftAxisX.posAbsolute[4] )
      I_Contact( "Unit1.Em5.ControlNodes".cm.command.transferPnPLeftAxisX.posAbsolute[5] )
      I_Contact( "Unit1.Em5.ControlNodes".cm.command.transferPnPLeftAxisX.posAbsolute[6] )
      I_Contact( "Unit1.Em5.ControlNodes".cm.command.transferPnPLeftAxisX.posAbsolute[7] )
      Not()
      Coil( "Unit1.Em5.ControlNodes".cm.command.transferPnPLeftAxisX.posAbsoluteSummary )
   END_RUNG
   // the same network as SCL:
   "Unit1.Em5.ControlNodes".cm.command.transferPnPLeftAxisX.posAbsoluteSummary := NOT (NOT "Unit1.Em5.ControlNodes".cm.command.transferPnPLeftAxisX.posAbsolute[0] AND NOT "Unit1.Em5.ControlNodes".cm.command.transferPnPLeftAxisX.posAbsolute[1] AND NOT "Unit1.Em5.ControlNodes".cm.command.transferPnPLeftAxisX.posAbsolute[2] AND NOT "Unit1.Em5.ControlNodes".cm.command.transferPnPLeftAxisX.posAbsolute[3] AND NOT "Unit1.Em5.ControlNodes".cm.command.transferPnPLeftAxisX.posAbsolute[4] AND NOT "Unit1.Em5.ControlNodes".cm.command.transferPnPLeftAxisX.posAbsolute[5] AND NOT "Unit1.Em5.ControlNodes".cm.command.transferPnPLeftAxisX.posAbsolute[6] AND NOT "Unit1.Em5.ControlNodes".cm.command.transferPnPLeftAxisX.posAbsolute[7]);
END_REGION

REGION Network 106: Transfer P&P Left AxisX Position Absolute Position
   RUNG wire#powerrail
      Contact( "Unit1.Em5.ControlNodes".cm.command.transferPnPLeftAxisX.posAbsoluteSummary )
      Coil( "Unit1.Em5.ControlNodes".cmTransferPnPLeftAxisX.commands.posAbsolute )
   END_RUNG
   // the same network as SCL:
   "Unit1.Em5.ControlNodes".cmTransferPnPLeftAxisX.commands.posAbsolute := "Unit1.Em5.ControlNodes".cm.command.transferPnPLeftAxisX.posAbsoluteSummary;
END_REGION

REGION Network 107: Transfer P&P Left AxisX Interlock Summary
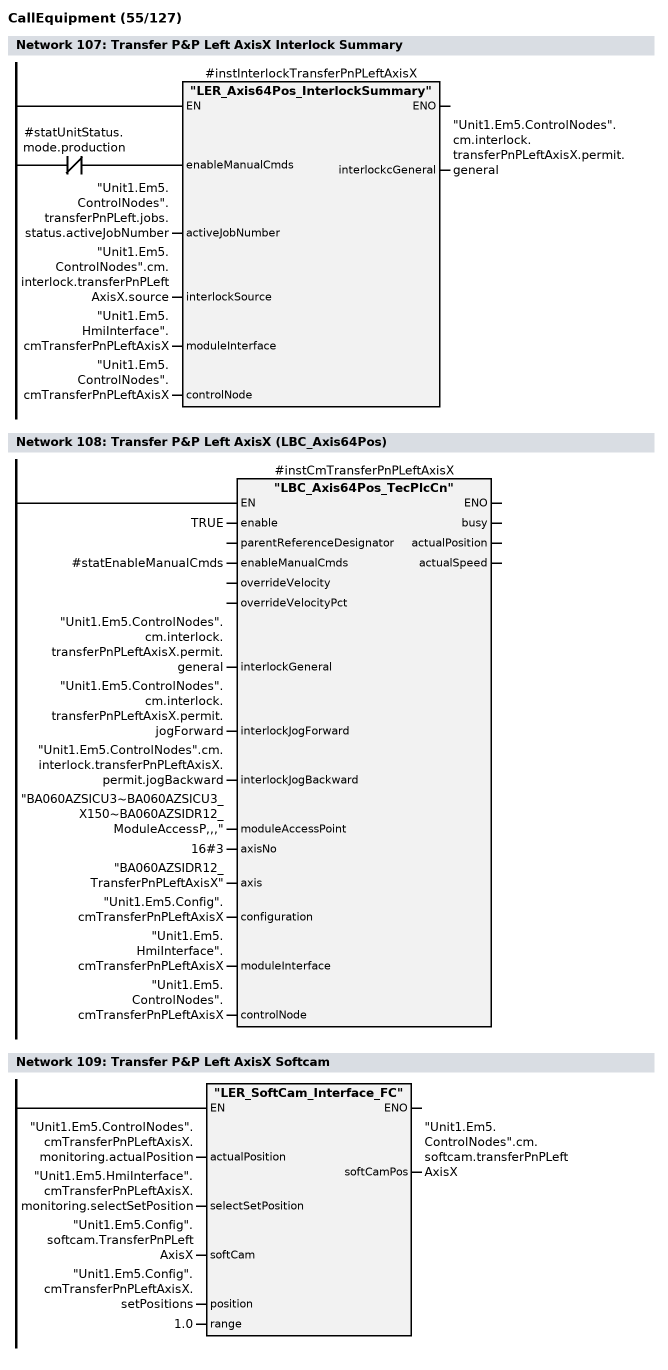
   RUNG wire#powerrail
      #instInterlockTransferPnPLeftAxisX(enableManualCmds := wire#w1, activeJobNumber := "Unit1.Em5.ControlNodes".transferPnPLeft.jobs.status.activeJobNumber, interlockSource := "Unit1.Em5.ControlNodes".cm.interlock.transferPnPLeftAxisX.source, moduleInterface := "Unit1.Em5.HmiInterface".cmTransferPnPLeftAxisX, controlNode := "Unit1.Em5.ControlNodes".cmTransferPnPLeftAxisX, interlockcGeneral => "Unit1.Em5.ControlNodes".cm.interlock.transferPnPLeftAxisX.permit.general)
   END_RUNG
   RUNG wire#powerrail
      I_Contact( #statUnitStatus.mode.production )
   END_RUNG wire#w1
   // the same network as SCL:
   #instInterlockTransferPnPLeftAxisX(enableManualCmds := NOT #statUnitStatus.mode.production,   // "LER_Axis64Pos_InterlockSummary"
                           activeJobNumber := "Unit1.Em5.ControlNodes".transferPnPLeft.jobs.status.activeJobNumber,
                           interlockSource := "Unit1.Em5.ControlNodes".cm.interlock.transferPnPLeftAxisX.source,
                           moduleInterface := "Unit1.Em5.HmiInterface".cmTransferPnPLeftAxisX,
                           controlNode := "Unit1.Em5.ControlNodes".cmTransferPnPLeftAxisX,
                           interlockcGeneral => "Unit1.Em5.ControlNodes".cm.interlock.transferPnPLeftAxisX.permit.general);
END_REGION

REGION Network 108: Transfer P&P Left AxisX (LBC_Axis64Pos)
   RUNG wire#powerrail
      #instCmTransferPnPLeftAxisX(enable := TRUE, parentReferenceDesignator :=, enableManualCmds := #statEnableManualCmds, overrideVelocity :=, overrideVelocityPct :=, interlockGeneral := "Unit1.Em5.ControlNodes".cm.interlock.transferPnPLeftAxisX.permit.general, interlockJogForward := "Unit1.Em5.ControlNodes".cm.interlock.transferPnPLeftAxisX.permit.jogForward, interlockJogBackward := "Unit1.Em5.ControlNodes".cm.interlock.transferPnPLeftAxisX.permit.jogBackward, moduleAccessPoint := "BA060AZSICU3~BA060AZSICU3_X150~BA060AZSIDR12_ModuleAccessP,,,", axisNo := 16#3, axis := "BA060AZSIDR12_TransferPnPLeftAxisX", configuration := "Unit1.Em5.Config".cmTransferPnPLeftAxisX, moduleInterface := "Unit1.Em5.HmiInterface".cmTransferPnPLeftAxisX, controlNode := "Unit1.Em5.ControlNodes".cmTransferPnPLeftAxisX, busy =>, actualPosition =>, actualSpeed =>)
   END_RUNG
   // the same network as SCL:
   #instCmTransferPnPLeftAxisX(enable := TRUE,   // "LBC_Axis64Pos_TecPlcCn"
                           enableManualCmds := #statEnableManualCmds,
                           interlockGeneral := "Unit1.Em5.ControlNodes".cm.interlock.transferPnPLeftAxisX.permit.general,
                           interlockJogForward := "Unit1.Em5.ControlNodes".cm.interlock.transferPnPLeftAxisX.permit.jogForward,
                           interlockJogBackward := "Unit1.Em5.ControlNodes".cm.interlock.transferPnPLeftAxisX.permit.jogBackward,
                           moduleAccessPoint := "BA060AZSICU3~BA060AZSICU3_X150~BA060AZSIDR12_ModuleAccessP,,,",
                           axisNo := 16#3,
                           axis := "BA060AZSIDR12_TransferPnPLeftAxisX",
                           configuration := "Unit1.Em5.Config".cmTransferPnPLeftAxisX,
                           moduleInterface := "Unit1.Em5.HmiInterface".cmTransferPnPLeftAxisX,
                           controlNode := "Unit1.Em5.ControlNodes".cmTransferPnPLeftAxisX);
END_REGION

REGION Network 109: Transfer P&P Left AxisX Softcam
   RUNG wire#powerrail
      "LER_SoftCam_Interface_FC"(actualPosition := "Unit1.Em5.ControlNodes".cmTransferPnPLeftAxisX.monitoring.actualPosition, selectSetPosition := "Unit1.Em5.HmiInterface".cmTransferPnPLeftAxisX.monitoring.selectSetPosition, softCam := "Unit1.Em5.Config".softcam.TransferPnPLeftAxisX, position := "Unit1.Em5.Config".cmTransferPnPLeftAxisX.setPositions, range := 1.0, softCamPos => "Unit1.Em5.ControlNodes".cm.softcam.transferPnPLeftAxisX)
   END_RUNG
   // the same network as SCL:
   "LER_SoftCam_Interface_FC"(actualPosition := "Unit1.Em5.ControlNodes".cmTransferPnPLeftAxisX.monitoring.actualPosition,
                           selectSetPosition := "Unit1.Em5.HmiInterface".cmTransferPnPLeftAxisX.monitoring.selectSetPosition,
                           softCam := "Unit1.Em5.Config".softcam.TransferPnPLeftAxisX,
                           position := "Unit1.Em5.Config".cmTransferPnPLeftAxisX.setPositions,
                           range := 1.0,
                           softCamPos => "Unit1.Em5.ControlNodes".cm.softcam.transferPnPLeftAxisX);
END_REGION

REGION Network 111: Transfer P&P Left Y-Axis Upload Actual Current And Torque Values
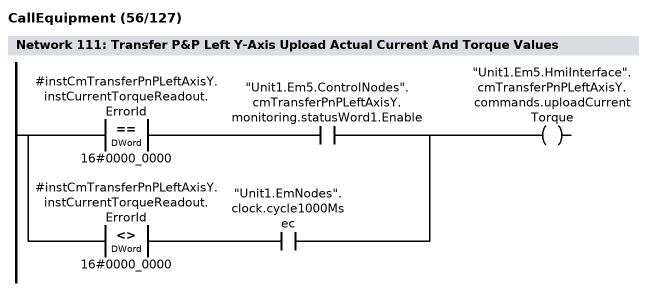
   RUNG wire#powerrail
      { S7_Templates := "SrcType := DWord" } EQ_Contact(in1 := #instCmTransferPnPLeftAxisY.instCurrentTorqueReadout.ErrorId, in2 := 16#0000_0000)
      Contact( "Unit1.Em5.ControlNodes".cmTransferPnPLeftAxisY.monitoring.statusWord1.Enable )
      wire#w1
      Coil( "Unit1.Em5.HmiInterface".cmTransferPnPLeftAxisY.commands.uploadCurrentTorque )
   END_RUNG
   RUNG wire#powerrail
      { S7_Templates := "SrcType := DWord" } NE_Contact(in1 := #instCmTransferPnPLeftAxisY.instCurrentTorqueReadout.ErrorId, in2 := 16#0000_0000)
      Contact( "Unit1.EmNodes".clock.cycle1000Msec )
   END_RUNG wire#w1
   // the same network as SCL:
   "Unit1.Em5.HmiInterface".cmTransferPnPLeftAxisY.commands.uploadCurrentTorque := ((#instCmTransferPnPLeftAxisY.instCurrentTorqueReadout.ErrorId = 16#0000_0000) AND "Unit1.Em5.ControlNodes".cmTransferPnPLeftAxisY.monitoring.statusWord1.Enable) OR ((#instCmTransferPnPLeftAxisY.instCurrentTorqueReadout.ErrorId <> 16#0000_0000) AND "Unit1.EmNodes".clock.cycle1000Msec);
END_REGION

REGION Network 112: Transfer PnP Left AxisY Home Interlock Condition
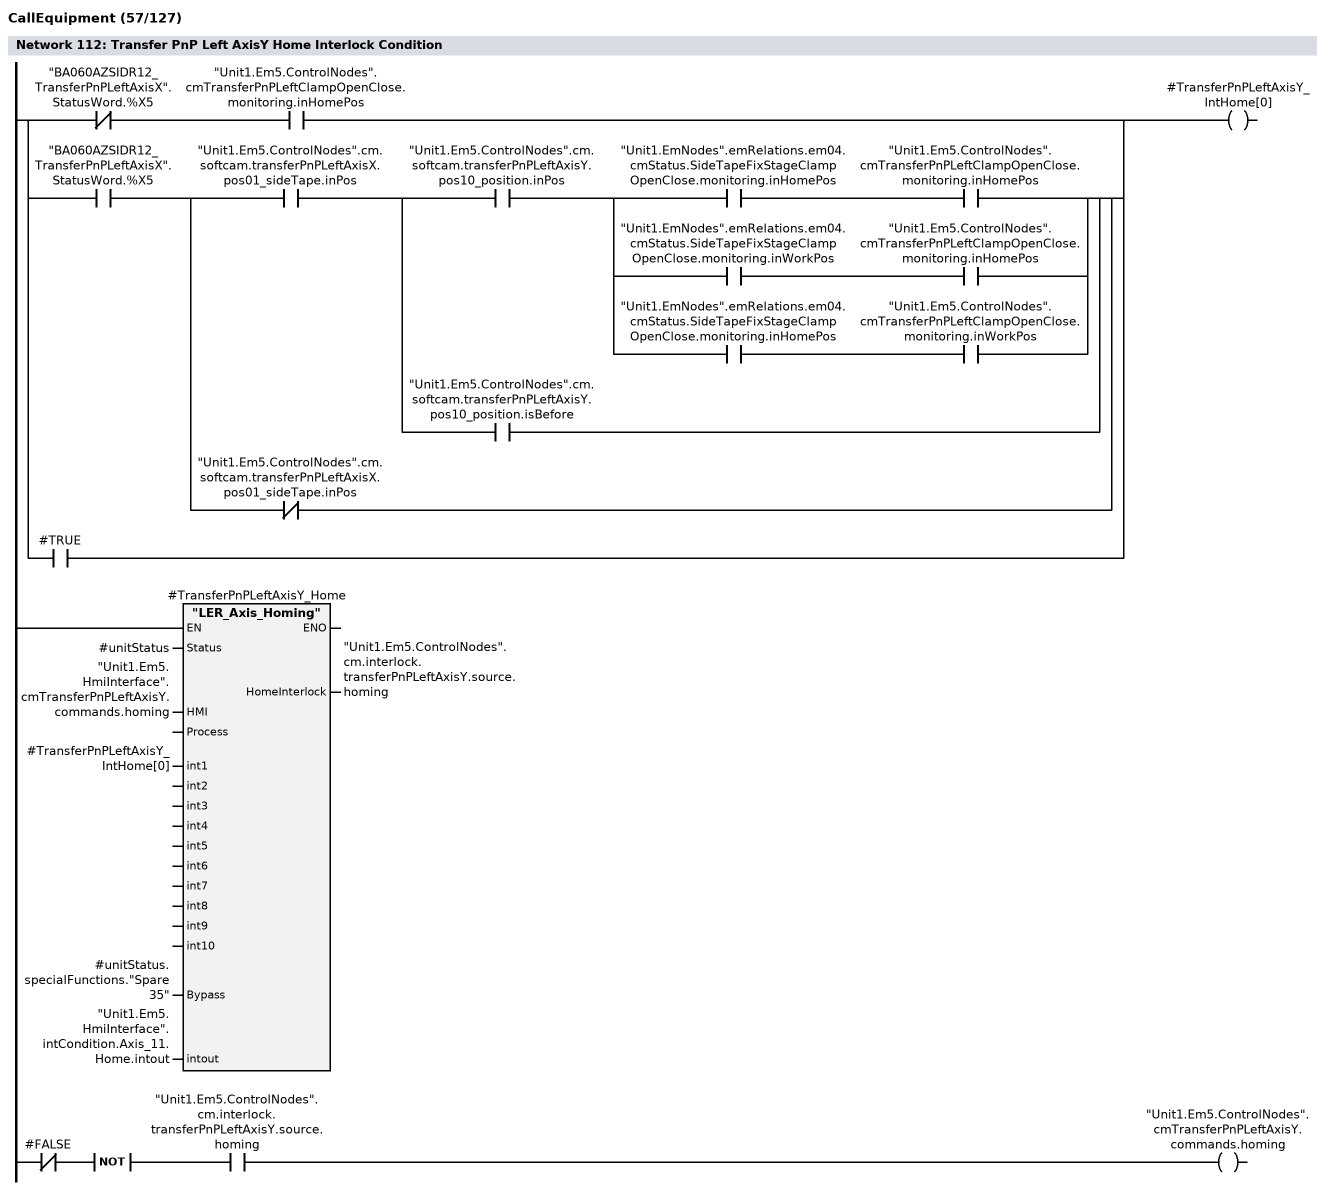
   RUNG wire#powerrail
      I_Contact( "BA060AZSIDR12_TransferPnPLeftAxisX".StatusWord.%X5 )
      Contact( "Unit1.Em5.ControlNodes".cmTransferPnPLeftClampOpenClose.monitoring.inHomePos )
      wire#w1
      Coil( #TransferPnPLeftAxisY_IntHome[0] )
   END_RUNG
   RUNG wire#powerrail
      Contact( "BA060AZSIDR12_TransferPnPLeftAxisX".StatusWord.%X5 )
      wire#w2
      Contact( "Unit1.Em5.ControlNodes".cm.softcam.transferPnPLeftAxisX.pos01_sideTape.inPos )
      wire#w3
      Contact( "Unit1.Em5.ControlNodes".cm.softcam.transferPnPLeftAxisY.pos10_position.inPos )
      wire#w4
      Contact( "Unit1.EmNodes".emRelations.em04.cmStatus.SideTapeFixStageClampOpenClose.monitoring.inHomePos )
      Contact( "Unit1.Em5.ControlNodes".cmTransferPnPLeftClampOpenClose.monitoring.inHomePos )
   END_RUNG wire#w1
   RUNG wire#w4
      Contact( "Unit1.EmNodes".emRelations.em04.cmStatus.SideTapeFixStageClampOpenClose.monitoring.inWorkPos )
      Contact( "Unit1.Em5.ControlNodes".cmTransferPnPLeftClampOpenClose.monitoring.inHomePos )
   END_RUNG wire#w1
   RUNG wire#w4
      Contact( "Unit1.EmNodes".emRelations.em04.cmStatus.SideTapeFixStageClampOpenClose.monitoring.inHomePos )
      Contact( "Unit1.Em5.ControlNodes".cmTransferPnPLeftClampOpenClose.monitoring.inWorkPos )
   END_RUNG wire#w1
   RUNG wire#w3
      Contact( "Unit1.Em5.ControlNodes".cm.softcam.transferPnPLeftAxisY.pos10_position.isBefore )
   END_RUNG wire#w1
   RUNG wire#w2
      I_Contact( "Unit1.Em5.ControlNodes".cm.softcam.transferPnPLeftAxisX.pos01_sideTape.inPos )
   END_RUNG wire#w1
   RUNG wire#powerrail
      Contact( #TRUE )
   END_RUNG wire#w1
   RUNG wire#powerrail
      #TransferPnPLeftAxisY_Home(Status := #unitStatus, HMI := "Unit1.Em5.HmiInterface".cmTransferPnPLeftAxisY.commands.homing, Process :=, int1 := #TransferPnPLeftAxisY_IntHome[0], int2 :=, int3 :=, int4 :=, int5 :=, int6 :=, int7 :=, int8 :=, int9 :=, int10 :=, Bypass := #unitStatus.specialFunctions."Spare 35", intout := "Unit1.Em5.HmiInterface".intCondition.Axis_11.Home.intout, HomeInterlock => "Unit1.Em5.ControlNodes".cm.interlock.transferPnPLeftAxisY.source.homing)
   END_RUNG
   RUNG wire#powerrail
      I_Contact( #FALSE )
      Not()
      Contact( "Unit1.Em5.ControlNodes".cm.interlock.transferPnPLeftAxisY.source.homing )
      Coil( "Unit1.Em5.ControlNodes".cmTransferPnPLeftAxisY.commands.homing )
   END_RUNG
   // the same network as SCL:
   #TransferPnPLeftAxisY_IntHome[0] := (NOT "BA060AZSIDR12_TransferPnPLeftAxisX".StatusWord.%X5 AND "Unit1.Em5.ControlNodes".cmTransferPnPLeftClampOpenClose.monitoring.inHomePos) OR ("BA060AZSIDR12_TransferPnPLeftAxisX".StatusWord.%X5 AND (("Unit1.Em5.ControlNodes".cm.softcam.transferPnPLeftAxisX.pos01_sideTape.inPos AND (("Unit1.Em5.ControlNodes".cm.softcam.transferPnPLeftAxisY.pos10_position.inPos AND (("Unit1.EmNodes".emRelations.em04.cmStatus.SideTapeFixStageClampOpenClose.monitoring.inHomePos AND "Unit1.Em5.ControlNodes".cmTransferPnPLeftClampOpenClose.monitoring.inHomePos) OR ("Unit1.EmNodes".emRelations.em04.cmStatus.SideTapeFixStageClampOpenClose.monitoring.inWorkPos AND "Unit1.Em5.ControlNodes".cmTransferPnPLeftClampOpenClose.monitoring.inHomePos) OR ("Unit1.EmNodes".emRelations.em04.cmStatus.SideTapeFixStageClampOpenClose.monitoring.inHomePos AND "Unit1.Em5.ControlNodes".cmTransferPnPLeftClampOpenClose.monitoring.inWorkPos))) OR "Unit1.Em5.ControlNodes".cm.softcam.transferPnPLeftAxisY.pos10_position.isBefore)) OR NOT "Unit1.Em5.ControlNodes".cm.softcam.transferPnPLeftAxisX.pos01_sideTape.inPos)) OR #TRUE;
   #TransferPnPLeftAxisY_Home(Status := #unitStatus,   // "LER_Axis_Homing"
                           HMI := "Unit1.Em5.HmiInterface".cmTransferPnPLeftAxisY.commands.homing,
                           int1 := #TransferPnPLeftAxisY_IntHome[0],
                           Bypass := #unitStatus.specialFunctions."Spare 35",
                           intout := "Unit1.Em5.HmiInterface".intCondition.Axis_11.Home.intout,
                           HomeInterlock => "Unit1.Em5.ControlNodes".cm.interlock.transferPnPLeftAxisY.source.homing);
   "Unit1.Em5.ControlNodes".cmTransferPnPLeftAxisY.commands.homing := NOT (NOT #FALSE) AND "Unit1.Em5.ControlNodes".cm.interlock.transferPnPLeftAxisY.source.homing;
END_REGION

REGION Network 113: Transfer PnP Left AxisY JOG Interlock Condition
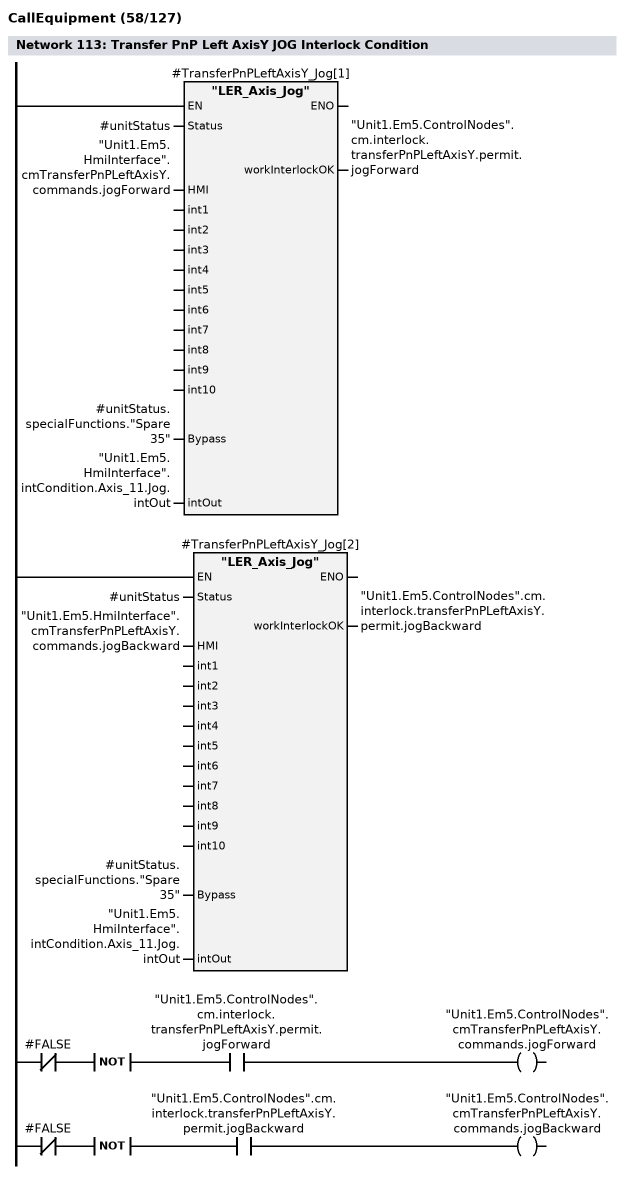
   RUNG wire#powerrail
      #TransferPnPLeftAxisY_Jog[1](Status := #unitStatus, HMI := "Unit1.Em5.HmiInterface".cmTransferPnPLeftAxisY.commands.jogForward, int1 :=, int2 :=, int3 :=, int4 :=, int5 :=, int6 :=, int7 :=, int8 :=, int9 :=, int10 :=, Bypass := #unitStatus.specialFunctions."Spare 35", intOut := "Unit1.Em5.HmiInterface".intCondition.Axis_11.Jog.intOut, workInterlockOK => "Unit1.Em5.ControlNodes".cm.interlock.transferPnPLeftAxisY.permit.jogForward)
   END_RUNG
   RUNG wire#powerrail
      #TransferPnPLeftAxisY_Jog[2](Status := #unitStatus, HMI := "Unit1.Em5.HmiInterface".cmTransferPnPLeftAxisY.commands.jogBackward, int1 :=, int2 :=, int3 :=, int4 :=, int5 :=, int6 :=, int7 :=, int8 :=, int9 :=, int10 :=, Bypass := #unitStatus.specialFunctions."Spare 35", intOut := "Unit1.Em5.HmiInterface".intCondition.Axis_11.Jog.intOut, workInterlockOK => "Unit1.Em5.ControlNodes".cm.interlock.transferPnPLeftAxisY.permit.jogBackward)
   END_RUNG
   RUNG wire#powerrail
      I_Contact( #FALSE )
      Not()
      Contact( "Unit1.Em5.ControlNodes".cm.interlock.transferPnPLeftAxisY.permit.jogForward )
      Coil( "Unit1.Em5.ControlNodes".cmTransferPnPLeftAxisY.commands.jogForward )
   END_RUNG
   RUNG wire#powerrail
      I_Contact( #FALSE )
      Not()
      Contact( "Unit1.Em5.ControlNodes".cm.interlock.transferPnPLeftAxisY.permit.jogBackward )
      Coil( "Unit1.Em5.ControlNodes".cmTransferPnPLeftAxisY.commands.jogBackward )
   END_RUNG
   // the same network as SCL:
   #TransferPnPLeftAxisY_Jog[1](Status := #unitStatus,   // "LER_Axis_Jog"
                           HMI := "Unit1.Em5.HmiInterface".cmTransferPnPLeftAxisY.commands.jogForward,
                           Bypass := #unitStatus.specialFunctions."Spare 35",
                           intOut := "Unit1.Em5.HmiInterface".intCondition.Axis_11.Jog.intOut,
                           workInterlockOK => "Unit1.Em5.ControlNodes".cm.interlock.transferPnPLeftAxisY.permit.jogForward);
   #TransferPnPLeftAxisY_Jog[2](Status := #unitStatus,   // "LER_Axis_Jog"
                           HMI := "Unit1.Em5.HmiInterface".cmTransferPnPLeftAxisY.commands.jogBackward,
                           Bypass := #unitStatus.specialFunctions."Spare 35",
                           intOut := "Unit1.Em5.HmiInterface".intCondition.Axis_11.Jog.intOut,
                           workInterlockOK => "Unit1.Em5.ControlNodes".cm.interlock.transferPnPLeftAxisY.permit.jogBackward);
   "Unit1.Em5.ControlNodes".cmTransferPnPLeftAxisY.commands.jogForward := NOT (NOT #FALSE) AND "Unit1.Em5.ControlNodes".cm.interlock.transferPnPLeftAxisY.permit.jogForward;
   "Unit1.Em5.ControlNodes".cmTransferPnPLeftAxisY.commands.jogBackward := NOT (NOT #FALSE) AND "Unit1.Em5.ControlNodes".cm.interlock.transferPnPLeftAxisY.permit.jogBackward;
END_REGION

REGION Network 114: Transfer PnP Left AxisY Position Absolute Position0
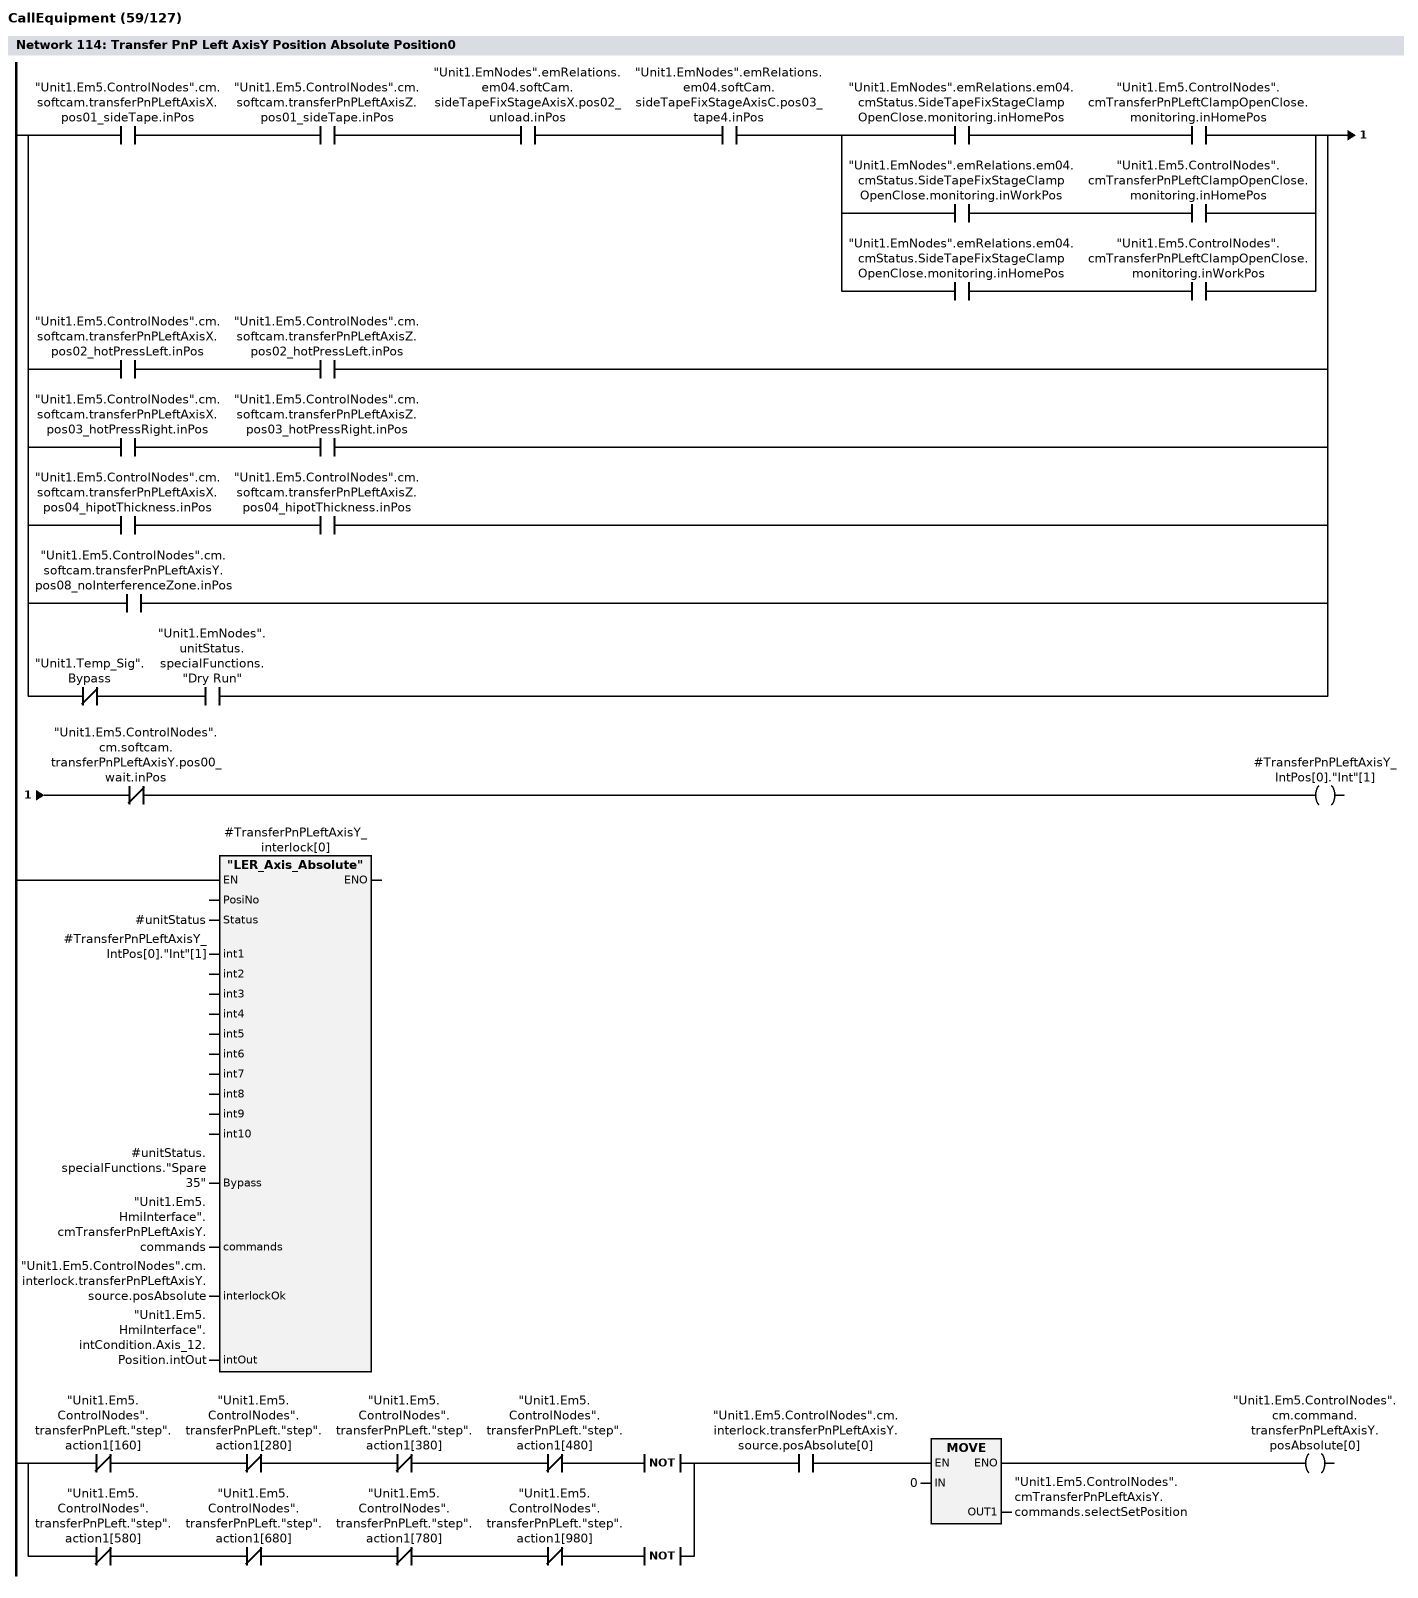
   RUNG wire#powerrail
      Contact( "Unit1.Em5.ControlNodes".cm.softcam.transferPnPLeftAxisX.pos01_sideTape.inPos )
      Contact( "Unit1.Em5.ControlNodes".cm.softcam.transferPnPLeftAxisZ.pos01_sideTape.inPos )
      Contact( "Unit1.EmNodes".emRelations.em04.softCam.sideTapeFixStageAxisX.pos02_unload.inPos )
      Contact( "Unit1.EmNodes".emRelations.em04.softCam.sideTapeFixStageAxisC.pos03_tape4.inPos )
      wire#w1
      Contact( "Unit1.EmNodes".emRelations.em04.cmStatus.SideTapeFixStageClampOpenClose.monitoring.inHomePos )
      Contact( "Unit1.Em5.ControlNodes".cmTransferPnPLeftClampOpenClose.monitoring.inHomePos )
      wire#w2
      I_Contact( "Unit1.Em5.ControlNodes".cm.softcam.transferPnPLeftAxisY.pos00_wait.inPos )
      Coil( #TransferPnPLeftAxisY_IntPos[0]."Int"[1] )
   END_RUNG
   RUNG wire#w1
      Contact( "Unit1.EmNodes".emRelations.em04.cmStatus.SideTapeFixStageClampOpenClose.monitoring.inWorkPos )
      Contact( "Unit1.Em5.ControlNodes".cmTransferPnPLeftClampOpenClose.monitoring.inHomePos )
   END_RUNG wire#w2
   RUNG wire#w1
      Contact( "Unit1.EmNodes".emRelations.em04.cmStatus.SideTapeFixStageClampOpenClose.monitoring.inHomePos )
      Contact( "Unit1.Em5.ControlNodes".cmTransferPnPLeftClampOpenClose.monitoring.inWorkPos )
   END_RUNG wire#w2
   RUNG wire#powerrail
      Contact( "Unit1.Em5.ControlNodes".cm.softcam.transferPnPLeftAxisX.pos02_hotPressLeft.inPos )
      Contact( "Unit1.Em5.ControlNodes".cm.softcam.transferPnPLeftAxisZ.pos02_hotPressLeft.inPos )
   END_RUNG wire#w2
   RUNG wire#powerrail
      Contact( "Unit1.Em5.ControlNodes".cm.softcam.transferPnPLeftAxisX.pos03_hotPressRight.inPos )
      Contact( "Unit1.Em5.ControlNodes".cm.softcam.transferPnPLeftAxisZ.pos03_hotPressRight.inPos )
   END_RUNG wire#w2
   RUNG wire#powerrail
      Contact( "Unit1.Em5.ControlNodes".cm.softcam.transferPnPLeftAxisX.pos04_hipotThickness.inPos )
      Contact( "Unit1.Em5.ControlNodes".cm.softcam.transferPnPLeftAxisZ.pos04_hipotThickness.inPos )
   END_RUNG wire#w2
   RUNG wire#powerrail
      Contact( "Unit1.Em5.ControlNodes".cm.softcam.transferPnPLeftAxisY.pos08_noInterferenceZone.inPos )
   END_RUNG wire#w2
   RUNG wire#powerrail
      I_Contact( "Unit1.Temp_Sig".Bypass )
      Contact( "Unit1.EmNodes".unitStatus.specialFunctions."Dry Run" )
   END_RUNG wire#w2
   RUNG wire#powerrail
      #TransferPnPLeftAxisY_interlock[0](PosiNo :=, Status := #unitStatus, int1 := #TransferPnPLeftAxisY_IntPos[0]."Int"[1], int2 :=, int3 :=, int4 :=, int5 :=, int6 :=, int7 :=, int8 :=, int9 :=, int10 :=, Bypass := #unitStatus.specialFunctions."Spare 35", commands := "Unit1.Em5.HmiInterface".cmTransferPnPLeftAxisY.commands, interlockOk := "Unit1.Em5.ControlNodes".cm.interlock.transferPnPLeftAxisY.source.posAbsolute, intOut := "Unit1.Em5.HmiInterface".intCondition.Axis_12.Position.intOut)
   END_RUNG
   RUNG wire#powerrail
      I_Contact( "Unit1.Em5.ControlNodes".transferPnPLeft."step".action1[160] )
      I_Contact( "Unit1.Em5.ControlNodes".transferPnPLeft."step".action1[280] )
      I_Contact( "Unit1.Em5.ControlNodes".transferPnPLeft."step".action1[380] )
      I_Contact( "Unit1.Em5.ControlNodes".transferPnPLeft."step".action1[480] )
      Not()
      wire#w3
      Contact( "Unit1.Em5.ControlNodes".cm.interlock.transferPnPLeftAxisY.source.posAbsolute[0] )
      Move(in := 0, out1 => "Unit1.Em5.ControlNodes".cmTransferPnPLeftAxisY.commands.selectSetPosition)
      Coil( "Unit1.Em5.ControlNodes".cm.command.transferPnPLeftAxisY.posAbsolute[0] )
   END_RUNG
   RUNG wire#powerrail
      I_Contact( "Unit1.Em5.ControlNodes".transferPnPLeft."step".action1[580] )
      I_Contact( "Unit1.Em5.ControlNodes".transferPnPLeft."step".action1[680] )
      I_Contact( "Unit1.Em5.ControlNodes".transferPnPLeft."step".action1[780] )
      I_Contact( "Unit1.Em5.ControlNodes".transferPnPLeft."step".action1[980] )
      Not()
   END_RUNG wire#w3
   // the same network as SCL:
   #TransferPnPLeftAxisY_IntPos[0]."Int"[1] := (("Unit1.Em5.ControlNodes".cm.softcam.transferPnPLeftAxisX.pos01_sideTape.inPos AND "Unit1.Em5.ControlNodes".cm.softcam.transferPnPLeftAxisZ.pos01_sideTape.inPos AND "Unit1.EmNodes".emRelations.em04.softCam.sideTapeFixStageAxisX.pos02_unload.inPos AND "Unit1.EmNodes".emRelations.em04.softCam.sideTapeFixStageAxisC.pos03_tape4.inPos AND (("Unit1.EmNodes".emRelations.em04.cmStatus.SideTapeFixStageClampOpenClose.monitoring.inHomePos AND "Unit1.Em5.ControlNodes".cmTransferPnPLeftClampOpenClose.monitoring.inHomePos) OR ("Unit1.EmNodes".emRelations.em04.cmStatus.SideTapeFixStageClampOpenClose.monitoring.inWorkPos AND "Unit1.Em5.ControlNodes".cmTransferPnPLeftClampOpenClose.monitoring.inHomePos) OR ("Unit1.EmNodes".emRelations.em04.cmStatus.SideTapeFixStageClampOpenClose.monitoring.inHomePos AND "Unit1.Em5.ControlNodes".cmTransferPnPLeftClampOpenClose.monitoring.inWorkPos))) OR ("Unit1.Em5.ControlNodes".cm.softcam.transferPnPLeftAxisX.pos02_hotPressLeft.inPos AND "Unit1.Em5.ControlNodes".cm.softcam.transferPnPLeftAxisZ.pos02_hotPressLeft.inPos) OR ("Unit1.Em5.ControlNodes".cm.softcam.transferPnPLeftAxisX.pos03_hotPressRight.inPos AND "Unit1.Em5.ControlNodes".cm.softcam.transferPnPLeftAxisZ.pos03_hotPressRight.inPos) OR ("Unit1.Em5.ControlNodes".cm.softcam.transferPnPLeftAxisX.pos04_hipotThickness.inPos AND "Unit1.Em5.ControlNodes".cm.softcam.transferPnPLeftAxisZ.pos04_hipotThickness.inPos) OR "Unit1.Em5.ControlNodes".cm.softcam.transferPnPLeftAxisY.pos08_noInterferenceZone.inPos OR (NOT "Unit1.Temp_Sig".Bypass AND "Unit1.EmNodes".unitStatus.specialFunctions."Dry Run")) AND NOT "Unit1.Em5.ControlNodes".cm.softcam.transferPnPLeftAxisY.pos00_wait.inPos;
   #TransferPnPLeftAxisY_interlock[0](Status := #unitStatus,   // "LER_Axis_Absolute"
                           int1 := #TransferPnPLeftAxisY_IntPos[0]."Int"[1],
                           Bypass := #unitStatus.specialFunctions."Spare 35",
                           commands := "Unit1.Em5.HmiInterface".cmTransferPnPLeftAxisY.commands,
                           interlockOk := "Unit1.Em5.ControlNodes".cm.interlock.transferPnPLeftAxisY.source.posAbsolute,
                           intOut := "Unit1.Em5.HmiInterface".intCondition.Axis_12.Position.intOut);
   #_w1 := (NOT (NOT "Unit1.Em5.ControlNodes".transferPnPLeft."step".action1[160] AND NOT "Unit1.Em5.ControlNodes".transferPnPLeft."step".action1[280] AND NOT "Unit1.Em5.ControlNodes".transferPnPLeft."step".action1[380] AND NOT "Unit1.Em5.ControlNodes".transferPnPLeft."step".action1[480]) OR NOT (NOT "Unit1.Em5.ControlNodes".transferPnPLeft."step".action1[580] AND NOT "Unit1.Em5.ControlNodes".transferPnPLeft."step".action1[680] AND NOT "Unit1.Em5.ControlNodes".transferPnPLeft."step".action1[780] AND NOT "Unit1.Em5.ControlNodes".transferPnPLeft."step".action1[980])) AND "Unit1.Em5.ControlNodes".cm.interlock.transferPnPLeftAxisY.source.posAbsolute[0];
   IF #_w1 THEN "Unit1.Em5.ControlNodes".cmTransferPnPLeftAxisY.commands.selectSetPosition := 0; END_IF;
   "Unit1.Em5.ControlNodes".cm.command.transferPnPLeftAxisY.posAbsolute[0] := #_w1;
END_REGION

REGION Network 115: Transfer PnP Left AxisY Position Absolute Position1
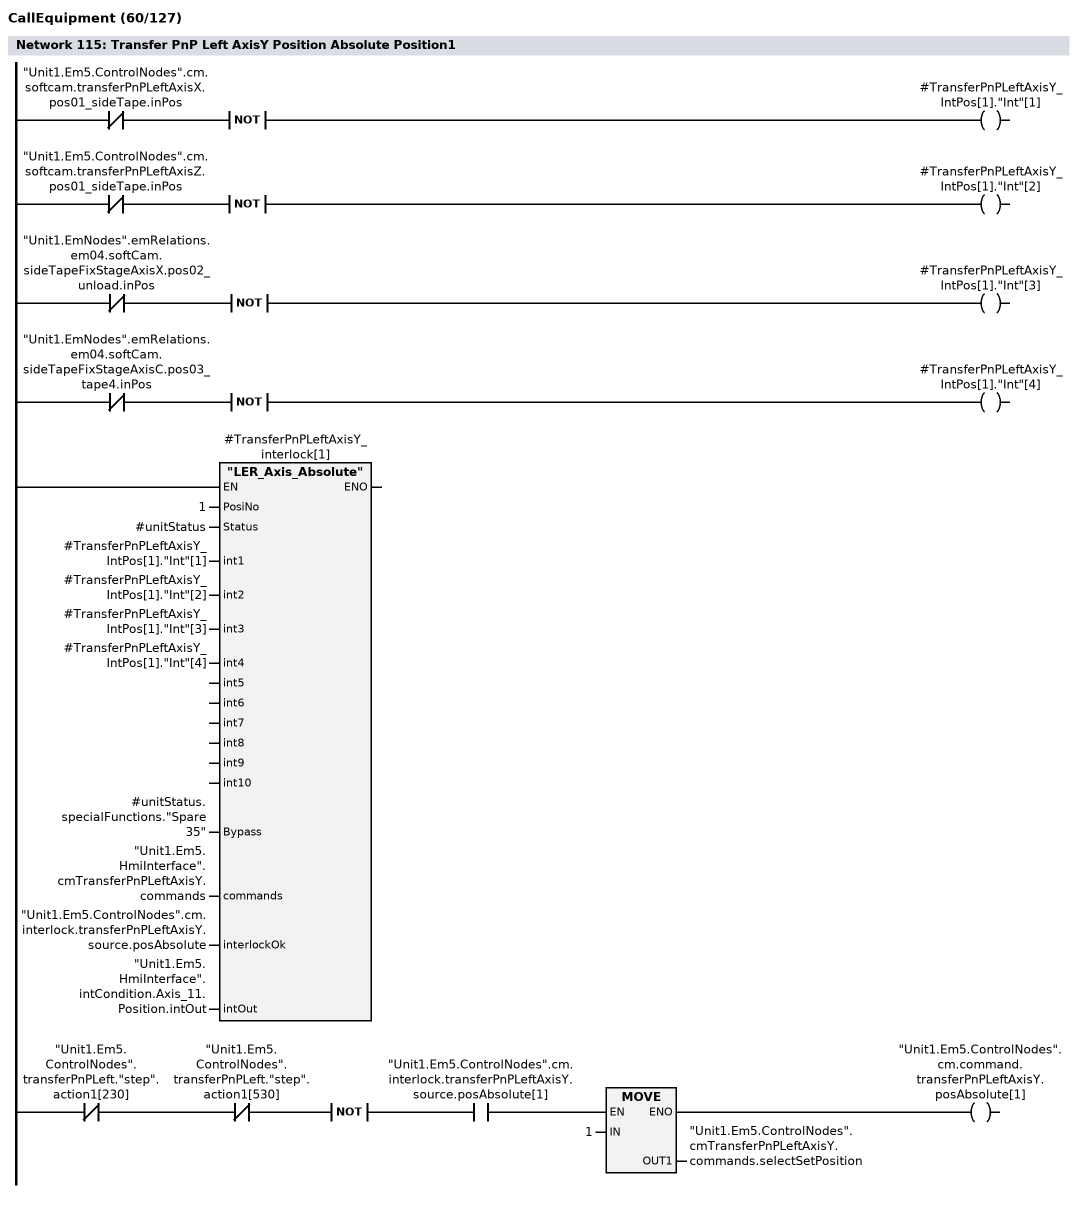
   RUNG wire#powerrail
      I_Contact( "Unit1.Em5.ControlNodes".cm.softcam.transferPnPLeftAxisX.pos01_sideTape.inPos )
      Not()
      Coil( #TransferPnPLeftAxisY_IntPos[1]."Int"[1] )
   END_RUNG
   RUNG wire#powerrail
      I_Contact( "Unit1.Em5.ControlNodes".cm.softcam.transferPnPLeftAxisZ.pos01_sideTape.inPos )
      Not()
      Coil( #TransferPnPLeftAxisY_IntPos[1]."Int"[2] )
   END_RUNG
   RUNG wire#powerrail
      I_Contact( "Unit1.EmNodes".emRelations.em04.softCam.sideTapeFixStageAxisX.pos02_unload.inPos )
      Not()
      Coil( #TransferPnPLeftAxisY_IntPos[1]."Int"[3] )
   END_RUNG
   RUNG wire#powerrail
      I_Contact( "Unit1.EmNodes".emRelations.em04.softCam.sideTapeFixStageAxisC.pos03_tape4.inPos )
      Not()
      Coil( #TransferPnPLeftAxisY_IntPos[1]."Int"[4] )
   END_RUNG
   RUNG wire#powerrail
      #TransferPnPLeftAxisY_interlock[1](PosiNo := 1, Status := #unitStatus, int1 := #TransferPnPLeftAxisY_IntPos[1]."Int"[1], int2 := #TransferPnPLeftAxisY_IntPos[1]."Int"[2], int3 := #TransferPnPLeftAxisY_IntPos[1]."Int"[3], int4 := #TransferPnPLeftAxisY_IntPos[1]."Int"[4], int5 :=, int6 :=, int7 :=, int8 :=, int9 :=, int10 :=, Bypass := #unitStatus.specialFunctions."Spare 35", commands := "Unit1.Em5.HmiInterface".cmTransferPnPLeftAxisY.commands, interlockOk := "Unit1.Em5.ControlNodes".cm.interlock.transferPnPLeftAxisY.source.posAbsolute, intOut := "Unit1.Em5.HmiInterface".intCondition.Axis_11.Position.intOut)
   END_RUNG
   RUNG wire#powerrail
      I_Contact( "Unit1.Em5.ControlNodes".transferPnPLeft."step".action1[230] )
      I_Contact( "Unit1.Em5.ControlNodes".transferPnPLeft."step".action1[530] )
      Not()
      Contact( "Unit1.Em5.ControlNodes".cm.interlock.transferPnPLeftAxisY.source.posAbsolute[1] )
      Move(in := 1, out1 => "Unit1.Em5.ControlNodes".cmTransferPnPLeftAxisY.commands.selectSetPosition)
      Coil( "Unit1.Em5.ControlNodes".cm.command.transferPnPLeftAxisY.posAbsolute[1] )
   END_RUNG
   // the same network as SCL:
   #TransferPnPLeftAxisY_IntPos[1]."Int"[1] := NOT (NOT "Unit1.Em5.ControlNodes".cm.softcam.transferPnPLeftAxisX.pos01_sideTape.inPos);
   #TransferPnPLeftAxisY_IntPos[1]."Int"[2] := NOT (NOT "Unit1.Em5.ControlNodes".cm.softcam.transferPnPLeftAxisZ.pos01_sideTape.inPos);
   #TransferPnPLeftAxisY_IntPos[1]."Int"[3] := NOT (NOT "Unit1.EmNodes".emRelations.em04.softCam.sideTapeFixStageAxisX.pos02_unload.inPos);
   #TransferPnPLeftAxisY_IntPos[1]."Int"[4] := NOT (NOT "Unit1.EmNodes".emRelations.em04.softCam.sideTapeFixStageAxisC.pos03_tape4.inPos);
   #TransferPnPLeftAxisY_interlock[1](PosiNo := 1,   // "LER_Axis_Absolute"
                           Status := #unitStatus,
                           int1 := #TransferPnPLeftAxisY_IntPos[1]."Int"[1],
                           int2 := #TransferPnPLeftAxisY_IntPos[1]."Int"[2],
                           int3 := #TransferPnPLeftAxisY_IntPos[1]."Int"[3],
                           int4 := #TransferPnPLeftAxisY_IntPos[1]."Int"[4],
                           Bypass := #unitStatus.specialFunctions."Spare 35",
                           commands := "Unit1.Em5.HmiInterface".cmTransferPnPLeftAxisY.commands,
                           interlockOk := "Unit1.Em5.ControlNodes".cm.interlock.transferPnPLeftAxisY.source.posAbsolute,
                           intOut := "Unit1.Em5.HmiInterface".intCondition.Axis_11.Position.intOut);
   #_w1 := NOT (NOT "Unit1.Em5.ControlNodes".transferPnPLeft."step".action1[230] AND NOT "Unit1.Em5.ControlNodes".transferPnPLeft."step".action1[530]) AND "Unit1.Em5.ControlNodes".cm.interlock.transferPnPLeftAxisY.source.posAbsolute[1];
   IF #_w1 THEN "Unit1.Em5.ControlNodes".cmTransferPnPLeftAxisY.commands.selectSetPosition := 1; END_IF;
   "Unit1.Em5.ControlNodes".cm.command.transferPnPLeftAxisY.posAbsolute[1] := #_w1;
END_REGION

REGION Network 116: Transfer PnP Left AxisY Position Absolute Position2
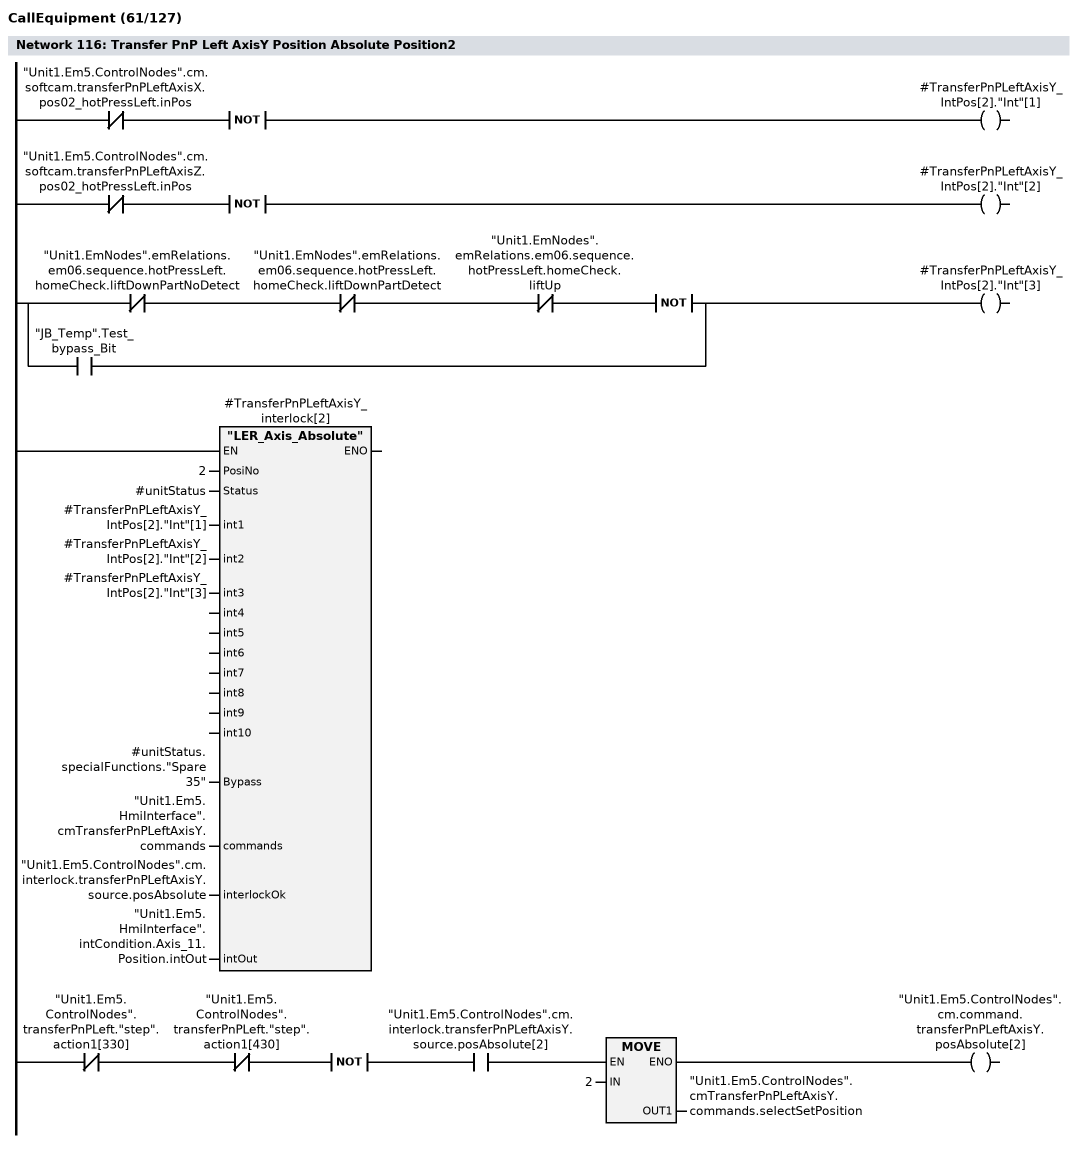
   RUNG wire#powerrail
      I_Contact( "Unit1.Em5.ControlNodes".cm.softcam.transferPnPLeftAxisX.pos02_hotPressLeft.inPos )
      Not()
      Coil( #TransferPnPLeftAxisY_IntPos[2]."Int"[1] )
   END_RUNG
   RUNG wire#powerrail
      I_Contact( "Unit1.Em5.ControlNodes".cm.softcam.transferPnPLeftAxisZ.pos02_hotPressLeft.inPos )
      Not()
      Coil( #TransferPnPLeftAxisY_IntPos[2]."Int"[2] )
   END_RUNG
   RUNG wire#powerrail
      I_Contact( "Unit1.EmNodes".emRelations.em06.sequence.hotPressLeft.homeCheck.liftDownPartNoDetect )
      I_Contact( "Unit1.EmNodes".emRelations.em06.sequence.hotPressLeft.homeCheck.liftDownPartDetect )
      I_Contact( "Unit1.EmNodes".emRelations.em06.sequence.hotPressLeft.homeCheck.liftUp )
      Not()
      wire#w1
      Coil( #TransferPnPLeftAxisY_IntPos[2]."Int"[3] )
   END_RUNG
   RUNG wire#powerrail
      Contact( "JB_Temp".Test_bypass_Bit )
   END_RUNG wire#w1
   RUNG wire#powerrail
      #TransferPnPLeftAxisY_interlock[2](PosiNo := 2, Status := #unitStatus, int1 := #TransferPnPLeftAxisY_IntPos[2]."Int"[1], int2 := #TransferPnPLeftAxisY_IntPos[2]."Int"[2], int3 := #TransferPnPLeftAxisY_IntPos[2]."Int"[3], int4 :=, int5 :=, int6 :=, int7 :=, int8 :=, int9 :=, int10 :=, Bypass := #unitStatus.specialFunctions."Spare 35", commands := "Unit1.Em5.HmiInterface".cmTransferPnPLeftAxisY.commands, interlockOk := "Unit1.Em5.ControlNodes".cm.interlock.transferPnPLeftAxisY.source.posAbsolute, intOut := "Unit1.Em5.HmiInterface".intCondition.Axis_11.Position.intOut)
   END_RUNG
   RUNG wire#powerrail
      I_Contact( "Unit1.Em5.ControlNodes".transferPnPLeft."step".action1[330] )
      I_Contact( "Unit1.Em5.ControlNodes".transferPnPLeft."step".action1[430] )
      Not()
      Contact( "Unit1.Em5.ControlNodes".cm.interlock.transferPnPLeftAxisY.source.posAbsolute[2] )
      Move(in := 2, out1 => "Unit1.Em5.ControlNodes".cmTransferPnPLeftAxisY.commands.selectSetPosition)
      Coil( "Unit1.Em5.ControlNodes".cm.command.transferPnPLeftAxisY.posAbsolute[2] )
   END_RUNG
   // the same network as SCL:
   #TransferPnPLeftAxisY_IntPos[2]."Int"[1] := NOT (NOT "Unit1.Em5.ControlNodes".cm.softcam.transferPnPLeftAxisX.pos02_hotPressLeft.inPos);
   #TransferPnPLeftAxisY_IntPos[2]."Int"[2] := NOT (NOT "Unit1.Em5.ControlNodes".cm.softcam.transferPnPLeftAxisZ.pos02_hotPressLeft.inPos);
   #TransferPnPLeftAxisY_IntPos[2]."Int"[3] := NOT (NOT "Unit1.EmNodes".emRelations.em06.sequence.hotPressLeft.homeCheck.liftDownPartNoDetect AND NOT "Unit1.EmNodes".emRelations.em06.sequence.hotPressLeft.homeCheck.liftDownPartDetect AND NOT "Unit1.EmNodes".emRelations.em06.sequence.hotPressLeft.homeCheck.liftUp) OR "JB_Temp".Test_bypass_Bit;
   #TransferPnPLeftAxisY_interlock[2](PosiNo := 2,   // "LER_Axis_Absolute"
                           Status := #unitStatus,
                           int1 := #TransferPnPLeftAxisY_IntPos[2]."Int"[1],
                           int2 := #TransferPnPLeftAxisY_IntPos[2]."Int"[2],
                           int3 := #TransferPnPLeftAxisY_IntPos[2]."Int"[3],
                           Bypass := #unitStatus.specialFunctions."Spare 35",
                           commands := "Unit1.Em5.HmiInterface".cmTransferPnPLeftAxisY.commands,
                           interlockOk := "Unit1.Em5.ControlNodes".cm.interlock.transferPnPLeftAxisY.source.posAbsolute,
                           intOut := "Unit1.Em5.HmiInterface".intCondition.Axis_11.Position.intOut);
   #_w1 := NOT (NOT "Unit1.Em5.ControlNodes".transferPnPLeft."step".action1[330] AND NOT "Unit1.Em5.ControlNodes".transferPnPLeft."step".action1[430]) AND "Unit1.Em5.ControlNodes".cm.interlock.transferPnPLeftAxisY.source.posAbsolute[2];
   IF #_w1 THEN "Unit1.Em5.ControlNodes".cmTransferPnPLeftAxisY.commands.selectSetPosition := 2; END_IF;
   "Unit1.Em5.ControlNodes".cm.command.transferPnPLeftAxisY.posAbsolute[2] := #_w1;
END_REGION

REGION Network 117: Transfer PnP Left AxisY Position Absolute Position3
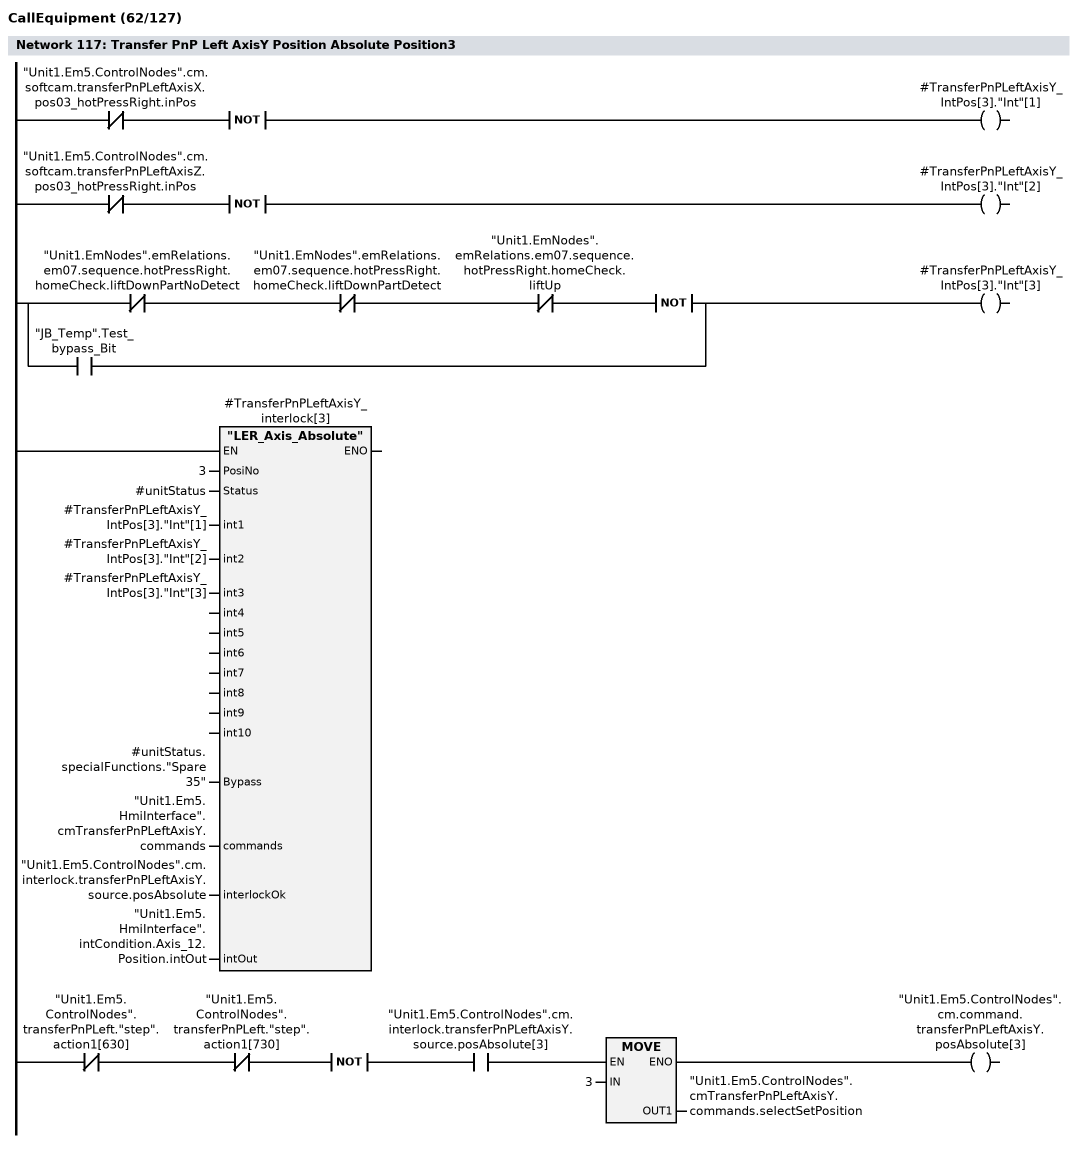
   RUNG wire#powerrail
      I_Contact( "Unit1.Em5.ControlNodes".cm.softcam.transferPnPLeftAxisX.pos03_hotPressRight.inPos )
      Not()
      Coil( #TransferPnPLeftAxisY_IntPos[3]."Int"[1] )
   END_RUNG
   RUNG wire#powerrail
      I_Contact( "Unit1.Em5.ControlNodes".cm.softcam.transferPnPLeftAxisZ.pos03_hotPressRight.inPos )
      Not()
      Coil( #TransferPnPLeftAxisY_IntPos[3]."Int"[2] )
   END_RUNG
   RUNG wire#powerrail
      I_Contact( "Unit1.EmNodes".emRelations.em07.sequence.hotPressRight.homeCheck.liftDownPartNoDetect )
      I_Contact( "Unit1.EmNodes".emRelations.em07.sequence.hotPressRight.homeCheck.liftDownPartDetect )
      I_Contact( "Unit1.EmNodes".emRelations.em07.sequence.hotPressRight.homeCheck.liftUp )
      Not()
      wire#w1
      Coil( #TransferPnPLeftAxisY_IntPos[3]."Int"[3] )
   END_RUNG
   RUNG wire#powerrail
      Contact( "JB_Temp".Test_bypass_Bit )
   END_RUNG wire#w1
   RUNG wire#powerrail
      #TransferPnPLeftAxisY_interlock[3](PosiNo := 3, Status := #unitStatus, int1 := #TransferPnPLeftAxisY_IntPos[3]."Int"[1], int2 := #TransferPnPLeftAxisY_IntPos[3]."Int"[2], int3 := #TransferPnPLeftAxisY_IntPos[3]."Int"[3], int4 :=, int5 :=, int6 :=, int7 :=, int8 :=, int9 :=, int10 :=, Bypass := #unitStatus.specialFunctions."Spare 35", commands := "Unit1.Em5.HmiInterface".cmTransferPnPLeftAxisY.commands, interlockOk := "Unit1.Em5.ControlNodes".cm.interlock.transferPnPLeftAxisY.source.posAbsolute, intOut := "Unit1.Em5.HmiInterface".intCondition.Axis_12.Position.intOut)
   END_RUNG
   RUNG wire#powerrail
      I_Contact( "Unit1.Em5.ControlNodes".transferPnPLeft."step".action1[630] )
      I_Contact( "Unit1.Em5.ControlNodes".transferPnPLeft."step".action1[730] )
      Not()
      Contact( "Unit1.Em5.ControlNodes".cm.interlock.transferPnPLeftAxisY.source.posAbsolute[3] )
      Move(in := 3, out1 => "Unit1.Em5.ControlNodes".cmTransferPnPLeftAxisY.commands.selectSetPosition)
      Coil( "Unit1.Em5.ControlNodes".cm.command.transferPnPLeftAxisY.posAbsolute[3] )
   END_RUNG
   // the same network as SCL:
   #TransferPnPLeftAxisY_IntPos[3]."Int"[1] := NOT (NOT "Unit1.Em5.ControlNodes".cm.softcam.transferPnPLeftAxisX.pos03_hotPressRight.inPos);
   #TransferPnPLeftAxisY_IntPos[3]."Int"[2] := NOT (NOT "Unit1.Em5.ControlNodes".cm.softcam.transferPnPLeftAxisZ.pos03_hotPressRight.inPos);
   #TransferPnPLeftAxisY_IntPos[3]."Int"[3] := NOT (NOT "Unit1.EmNodes".emRelations.em07.sequence.hotPressRight.homeCheck.liftDownPartNoDetect AND NOT "Unit1.EmNodes".emRelations.em07.sequence.hotPressRight.homeCheck.liftDownPartDetect AND NOT "Unit1.EmNodes".emRelations.em07.sequence.hotPressRight.homeCheck.liftUp) OR "JB_Temp".Test_bypass_Bit;
   #TransferPnPLeftAxisY_interlock[3](PosiNo := 3,   // "LER_Axis_Absolute"
                           Status := #unitStatus,
                           int1 := #TransferPnPLeftAxisY_IntPos[3]."Int"[1],
                           int2 := #TransferPnPLeftAxisY_IntPos[3]."Int"[2],
                           int3 := #TransferPnPLeftAxisY_IntPos[3]."Int"[3],
                           Bypass := #unitStatus.specialFunctions."Spare 35",
                           commands := "Unit1.Em5.HmiInterface".cmTransferPnPLeftAxisY.commands,
                           interlockOk := "Unit1.Em5.ControlNodes".cm.interlock.transferPnPLeftAxisY.source.posAbsolute,
                           intOut := "Unit1.Em5.HmiInterface".intCondition.Axis_12.Position.intOut);
   #_w1 := NOT (NOT "Unit1.Em5.ControlNodes".transferPnPLeft."step".action1[630] AND NOT "Unit1.Em5.ControlNodes".transferPnPLeft."step".action1[730]) AND "Unit1.Em5.ControlNodes".cm.interlock.transferPnPLeftAxisY.source.posAbsolute[3];
   IF #_w1 THEN "Unit1.Em5.ControlNodes".cmTransferPnPLeftAxisY.commands.selectSetPosition := 3; END_IF;
   "Unit1.Em5.ControlNodes".cm.command.transferPnPLeftAxisY.posAbsolute[3] := #_w1;
END_REGION

REGION Network 118: Transfer PnP Left AxisY Position Absolute Position4
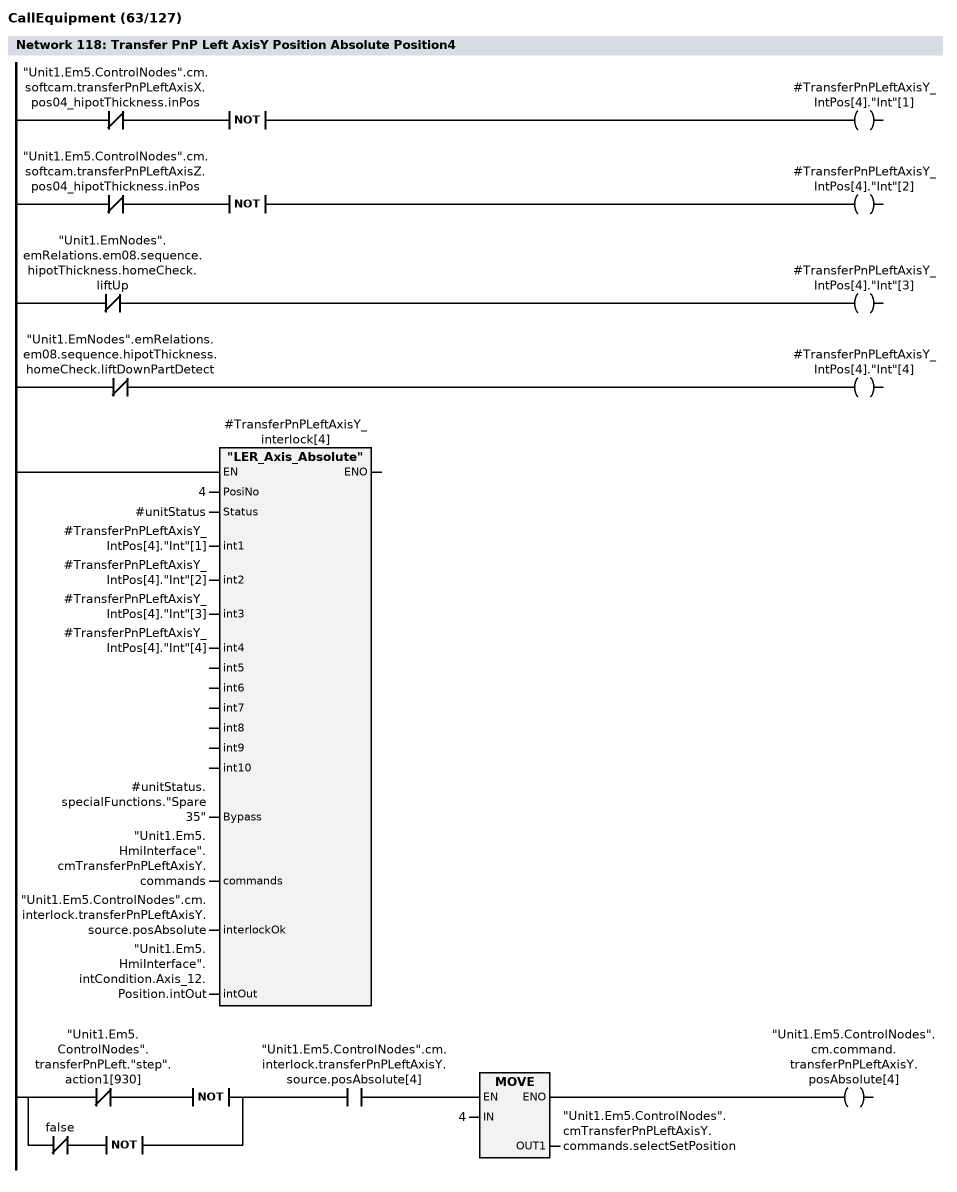
   RUNG wire#powerrail
      I_Contact( "Unit1.Em5.ControlNodes".cm.softcam.transferPnPLeftAxisX.pos04_hipotThickness.inPos )
      Not()
      Coil( #TransferPnPLeftAxisY_IntPos[4]."Int"[1] )
   END_RUNG
   RUNG wire#powerrail
      I_Contact( "Unit1.Em5.ControlNodes".cm.softcam.transferPnPLeftAxisZ.pos04_hipotThickness.inPos )
      Not()
      Coil( #TransferPnPLeftAxisY_IntPos[4]."Int"[2] )
   END_RUNG
   RUNG wire#powerrail
      I_Contact( "Unit1.EmNodes".emRelations.em08.sequence.hipotThickness.homeCheck.liftUp )
      Coil( #TransferPnPLeftAxisY_IntPos[4]."Int"[3] )
   END_RUNG
   RUNG wire#powerrail
      I_Contact( "Unit1.EmNodes".emRelations.em08.sequence.hipotThickness.homeCheck.liftDownPartDetect )
      Coil( #TransferPnPLeftAxisY_IntPos[4]."Int"[4] )
   END_RUNG
   RUNG wire#powerrail
      #TransferPnPLeftAxisY_interlock[4](PosiNo := 4, Status := #unitStatus, int1 := #TransferPnPLeftAxisY_IntPos[4]."Int"[1], int2 := #TransferPnPLeftAxisY_IntPos[4]."Int"[2], int3 := #TransferPnPLeftAxisY_IntPos[4]."Int"[3], int4 := #TransferPnPLeftAxisY_IntPos[4]."Int"[4], int5 :=, int6 :=, int7 :=, int8 :=, int9 :=, int10 :=, Bypass := #unitStatus.specialFunctions."Spare 35", commands := "Unit1.Em5.HmiInterface".cmTransferPnPLeftAxisY.commands, interlockOk := "Unit1.Em5.ControlNodes".cm.interlock.transferPnPLeftAxisY.source.posAbsolute, intOut := "Unit1.Em5.HmiInterface".intCondition.Axis_12.Position.intOut)
   END_RUNG
   RUNG wire#powerrail
      I_Contact( "Unit1.Em5.ControlNodes".transferPnPLeft."step".action1[930] )
      Not()
      wire#w1
      Contact( "Unit1.Em5.ControlNodes".cm.interlock.transferPnPLeftAxisY.source.posAbsolute[4] )
      Move(in := 4, out1 => "Unit1.Em5.ControlNodes".cmTransferPnPLeftAxisY.commands.selectSetPosition)
      Coil( "Unit1.Em5.ControlNodes".cm.command.transferPnPLeftAxisY.posAbsolute[4] )
   END_RUNG
   RUNG wire#powerrail
      I_Contact( false )
      Not()
   END_RUNG wire#w1
   // the same network as SCL:
   #TransferPnPLeftAxisY_IntPos[4]."Int"[1] := NOT (NOT "Unit1.Em5.ControlNodes".cm.softcam.transferPnPLeftAxisX.pos04_hipotThickness.inPos);
   #TransferPnPLeftAxisY_IntPos[4]."Int"[2] := NOT (NOT "Unit1.Em5.ControlNodes".cm.softcam.transferPnPLeftAxisZ.pos04_hipotThickness.inPos);
   #TransferPnPLeftAxisY_IntPos[4]."Int"[3] := NOT "Unit1.EmNodes".emRelations.em08.sequence.hipotThickness.homeCheck.liftUp;
   #TransferPnPLeftAxisY_IntPos[4]."Int"[4] := NOT "Unit1.EmNodes".emRelations.em08.sequence.hipotThickness.homeCheck.liftDownPartDetect;
   #TransferPnPLeftAxisY_interlock[4](PosiNo := 4,   // "LER_Axis_Absolute"
                           Status := #unitStatus,
                           int1 := #TransferPnPLeftAxisY_IntPos[4]."Int"[1],
                           int2 := #TransferPnPLeftAxisY_IntPos[4]."Int"[2],
                           int3 := #TransferPnPLeftAxisY_IntPos[4]."Int"[3],
                           int4 := #TransferPnPLeftAxisY_IntPos[4]."Int"[4],
                           Bypass := #unitStatus.specialFunctions."Spare 35",
                           commands := "Unit1.Em5.HmiInterface".cmTransferPnPLeftAxisY.commands,
                           interlockOk := "Unit1.Em5.ControlNodes".cm.interlock.transferPnPLeftAxisY.source.posAbsolute,
                           intOut := "Unit1.Em5.HmiInterface".intCondition.Axis_12.Position.intOut);
   #_w1 := (NOT (NOT "Unit1.Em5.ControlNodes".transferPnPLeft."step".action1[930]) OR NOT (NOT false)) AND "Unit1.Em5.ControlNodes".cm.interlock.transferPnPLeftAxisY.source.posAbsolute[4];
   IF #_w1 THEN "Unit1.Em5.ControlNodes".cmTransferPnPLeftAxisY.commands.selectSetPosition := 4; END_IF;
   "Unit1.Em5.ControlNodes".cm.command.transferPnPLeftAxisY.posAbsolute[4] := #_w1;
END_REGION

REGION Network 119: Transfer PnP Left AxisY Position Absolute Position5
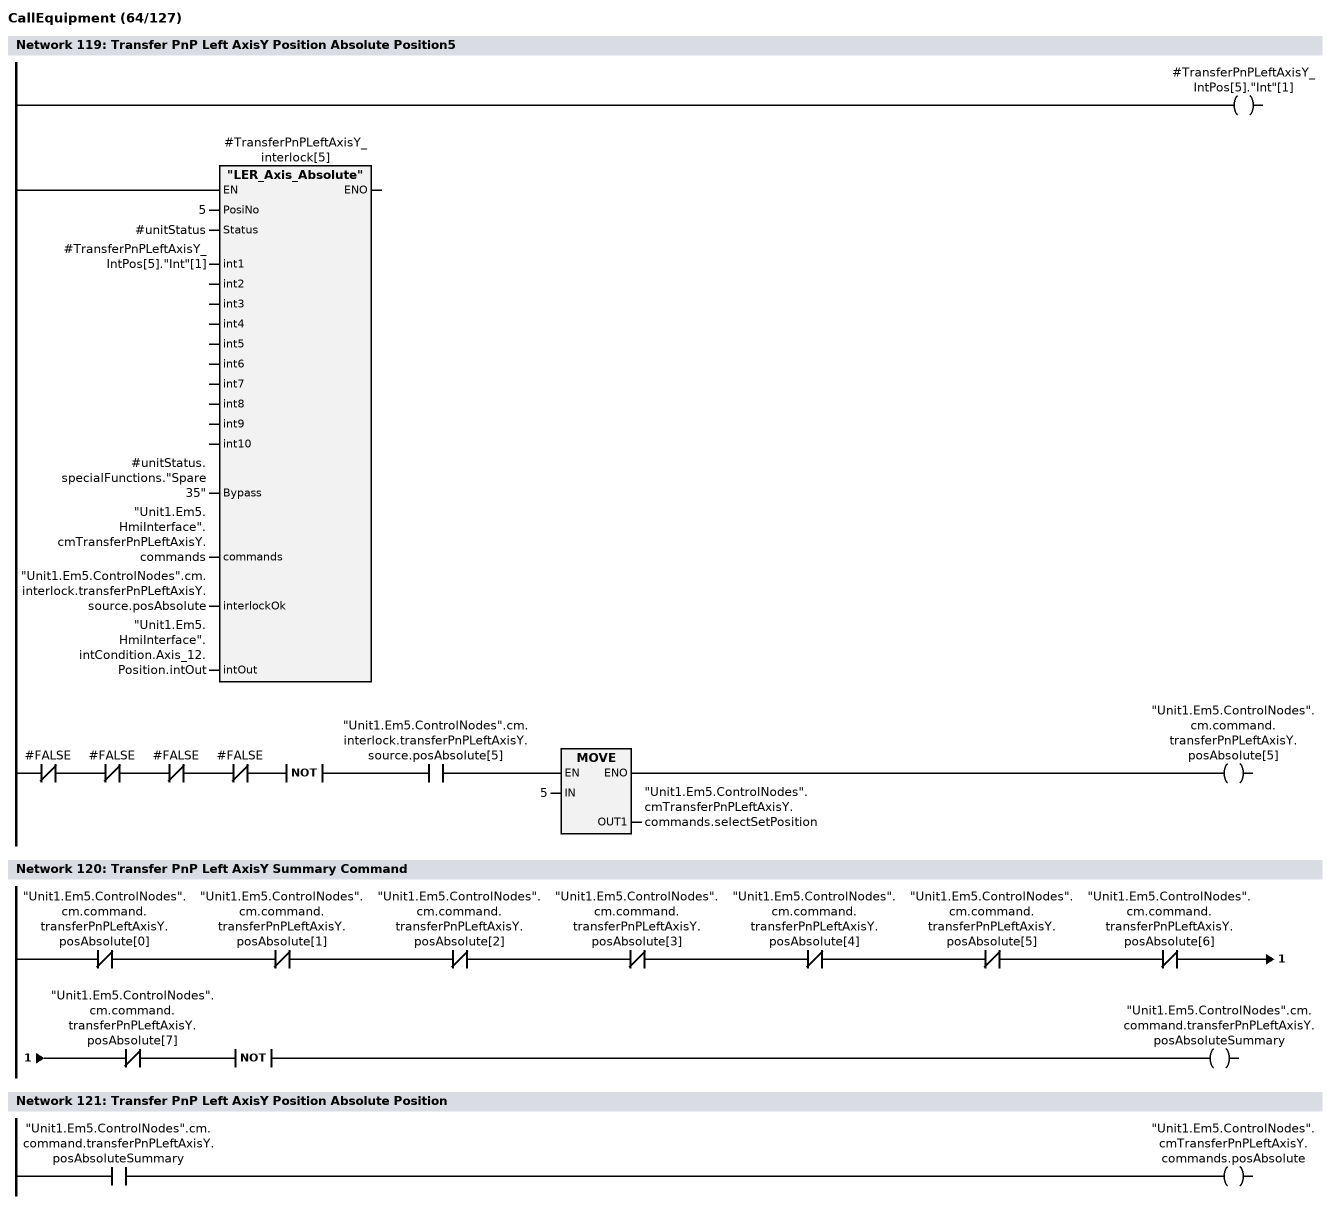
   RUNG wire#powerrail
      Coil( #TransferPnPLeftAxisY_IntPos[5]."Int"[1] )
   END_RUNG
   RUNG wire#powerrail
      #TransferPnPLeftAxisY_interlock[5](PosiNo := 5, Status := #unitStatus, int1 := #TransferPnPLeftAxisY_IntPos[5]."Int"[1], int2 :=, int3 :=, int4 :=, int5 :=, int6 :=, int7 :=, int8 :=, int9 :=, int10 :=, Bypass := #unitStatus.specialFunctions."Spare 35", commands := "Unit1.Em5.HmiInterface".cmTransferPnPLeftAxisY.commands, interlockOk := "Unit1.Em5.ControlNodes".cm.interlock.transferPnPLeftAxisY.source.posAbsolute, intOut := "Unit1.Em5.HmiInterface".intCondition.Axis_12.Position.intOut)
   END_RUNG
   RUNG wire#powerrail
      I_Contact( #FALSE )
      I_Contact( #FALSE )
      I_Contact( #FALSE )
      I_Contact( #FALSE )
      Not()
      Contact( "Unit1.Em5.ControlNodes".cm.interlock.transferPnPLeftAxisY.source.posAbsolute[5] )
      Move(in := 5, out1 => "Unit1.Em5.ControlNodes".cmTransferPnPLeftAxisY.commands.selectSetPosition)
      Coil( "Unit1.Em5.ControlNodes".cm.command.transferPnPLeftAxisY.posAbsolute[5] )
   END_RUNG
   // the same network as SCL:
   #TransferPnPLeftAxisY_IntPos[5]."Int"[1] := TRUE;
   #TransferPnPLeftAxisY_interlock[5](PosiNo := 5,   // "LER_Axis_Absolute"
                           Status := #unitStatus,
                           int1 := #TransferPnPLeftAxisY_IntPos[5]."Int"[1],
                           Bypass := #unitStatus.specialFunctions."Spare 35",
                           commands := "Unit1.Em5.HmiInterface".cmTransferPnPLeftAxisY.commands,
                           interlockOk := "Unit1.Em5.ControlNodes".cm.interlock.transferPnPLeftAxisY.source.posAbsolute,
                           intOut := "Unit1.Em5.HmiInterface".intCondition.Axis_12.Position.intOut);
   #_w1 := NOT (NOT #FALSE AND NOT #FALSE AND NOT #FALSE AND NOT #FALSE) AND "Unit1.Em5.ControlNodes".cm.interlock.transferPnPLeftAxisY.source.posAbsolute[5];
   IF #_w1 THEN "Unit1.Em5.ControlNodes".cmTransferPnPLeftAxisY.commands.selectSetPosition := 5; END_IF;
   "Unit1.Em5.ControlNodes".cm.command.transferPnPLeftAxisY.posAbsolute[5] := #_w1;
END_REGION

REGION Network 120: Transfer PnP Left AxisY Summary Command
   RUNG wire#powerrail
      I_Contact( "Unit1.Em5.ControlNodes".cm.command.transferPnPLeftAxisY.posAbsolute[0] )
      I_Contact( "Unit1.Em5.ControlNodes".cm.command.transferPnPLeftAxisY.posAbsolute[1] )
      I_Contact( "Unit1.Em5.ControlNodes".cm.command.transferPnPLeftAxisY.posAbsolute[2] )
      I_Contact( "Unit1.Em5.ControlNodes".cm.command.transferPnPLeftAxisY.posAbsolute[3] )
      I_Contact( "Unit1.Em5.ControlNodes".cm.command.transferPnPLeftAxisY.posAbsolute[4] )
      I_Contact( "Unit1.Em5.ControlNodes".cm.command.transferPnPLeftAxisY.posAbsolute[5] )
      I_Contact( "Unit1.Em5.ControlNodes".cm.command.transferPnPLeftAxisY.posAbsolute[6] )
      I_Contact( "Unit1.Em5.ControlNodes".cm.command.transferPnPLeftAxisY.posAbsolute[7] )
      Not()
      Coil( "Unit1.Em5.ControlNodes".cm.command.transferPnPLeftAxisY.posAbsoluteSummary )
   END_RUNG
   // the same network as SCL:
   "Unit1.Em5.ControlNodes".cm.command.transferPnPLeftAxisY.posAbsoluteSummary := NOT (NOT "Unit1.Em5.ControlNodes".cm.command.transferPnPLeftAxisY.posAbsolute[0] AND NOT "Unit1.Em5.ControlNodes".cm.command.transferPnPLeftAxisY.posAbsolute[1] AND NOT "Unit1.Em5.ControlNodes".cm.command.transferPnPLeftAxisY.posAbsolute[2] AND NOT "Unit1.Em5.ControlNodes".cm.command.transferPnPLeftAxisY.posAbsolute[3] AND NOT "Unit1.Em5.ControlNodes".cm.command.transferPnPLeftAxisY.posAbsolute[4] AND NOT "Unit1.Em5.ControlNodes".cm.command.transferPnPLeftAxisY.posAbsolute[5] AND NOT "Unit1.Em5.ControlNodes".cm.command.transferPnPLeftAxisY.posAbsolute[6] AND NOT "Unit1.Em5.ControlNodes".cm.command.transferPnPLeftAxisY.posAbsolute[7]);
END_REGION

REGION Network 121: Transfer PnP Left AxisY Position Absolute Position
   RUNG wire#powerrail
      Contact( "Unit1.Em5.ControlNodes".cm.command.transferPnPLeftAxisY.posAbsoluteSummary )
      Coil( "Unit1.Em5.ControlNodes".cmTransferPnPLeftAxisY.commands.posAbsolute )
   END_RUNG
   // the same network as SCL:
   "Unit1.Em5.ControlNodes".cmTransferPnPLeftAxisY.commands.posAbsolute := "Unit1.Em5.ControlNodes".cm.command.transferPnPLeftAxisY.posAbsoluteSummary;
END_REGION

REGION Network 122: Transfer PnP Left AxisY Interlock Summary
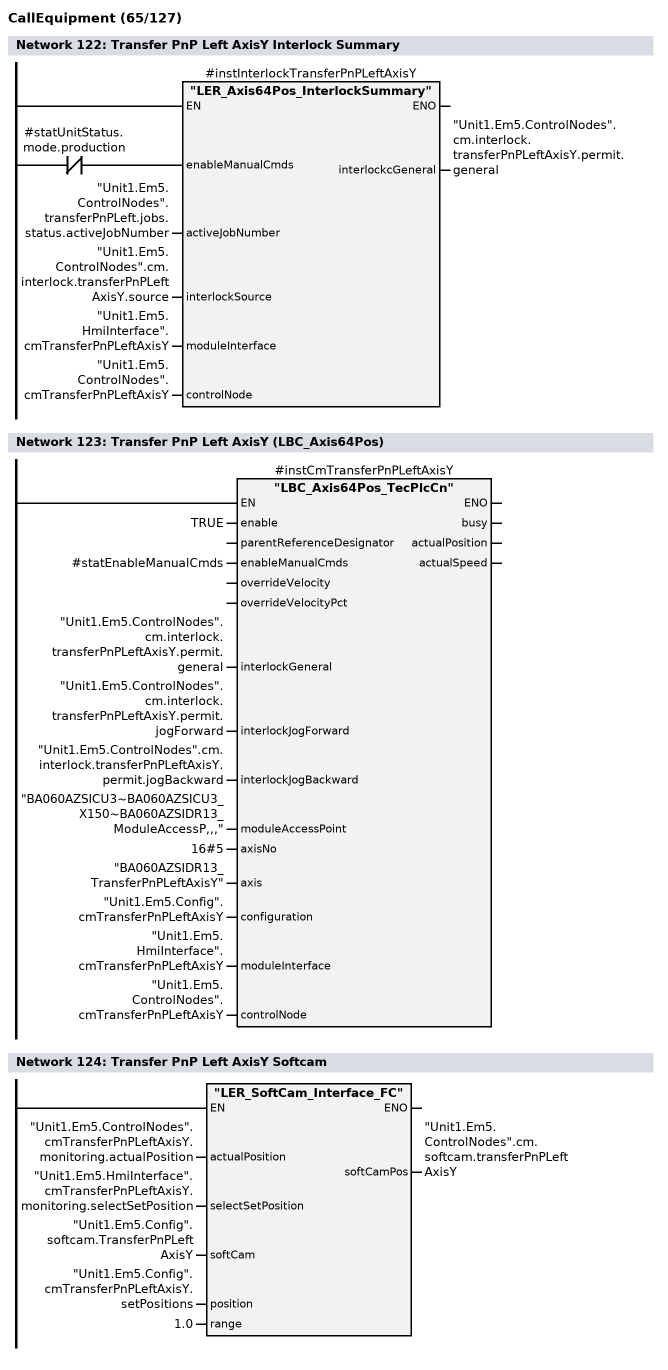
   RUNG wire#powerrail
      #instInterlockTransferPnPLeftAxisY(enableManualCmds := wire#w1, activeJobNumber := "Unit1.Em5.ControlNodes".transferPnPLeft.jobs.status.activeJobNumber, interlockSource := "Unit1.Em5.ControlNodes".cm.interlock.transferPnPLeftAxisY.source, moduleInterface := "Unit1.Em5.HmiInterface".cmTransferPnPLeftAxisY, controlNode := "Unit1.Em5.ControlNodes".cmTransferPnPLeftAxisY, interlockcGeneral => "Unit1.Em5.ControlNodes".cm.interlock.transferPnPLeftAxisY.permit.general)
   END_RUNG
   RUNG wire#powerrail
      I_Contact( #statUnitStatus.mode.production )
   END_RUNG wire#w1
   // the same network as SCL:
   #instInterlockTransferPnPLeftAxisY(enableManualCmds := NOT #statUnitStatus.mode.production,   // "LER_Axis64Pos_InterlockSummary"
                           activeJobNumber := "Unit1.Em5.ControlNodes".transferPnPLeft.jobs.status.activeJobNumber,
                           interlockSource := "Unit1.Em5.ControlNodes".cm.interlock.transferPnPLeftAxisY.source,
                           moduleInterface := "Unit1.Em5.HmiInterface".cmTransferPnPLeftAxisY,
                           controlNode := "Unit1.Em5.ControlNodes".cmTransferPnPLeftAxisY,
                           interlockcGeneral => "Unit1.Em5.ControlNodes".cm.interlock.transferPnPLeftAxisY.permit.general);
END_REGION

REGION Network 123: Transfer PnP Left AxisY (LBC_Axis64Pos)
   RUNG wire#powerrail
      #instCmTransferPnPLeftAxisY(enable := TRUE, parentReferenceDesignator :=, enableManualCmds := #statEnableManualCmds, overrideVelocity :=, overrideVelocityPct :=, interlockGeneral := "Unit1.Em5.ControlNodes".cm.interlock.transferPnPLeftAxisY.permit.general, interlockJogForward := "Unit1.Em5.ControlNodes".cm.interlock.transferPnPLeftAxisY.permit.jogForward, interlockJogBackward := "Unit1.Em5.ControlNodes".cm.interlock.transferPnPLeftAxisY.permit.jogBackward, moduleAccessPoint := "BA060AZSICU3~BA060AZSICU3_X150~BA060AZSIDR13_ModuleAccessP,,,", axisNo := 16#5, axis := "BA060AZSIDR13_TransferPnPLeftAxisY", configuration := "Unit1.Em5.Config".cmTransferPnPLeftAxisY, moduleInterface := "Unit1.Em5.HmiInterface".cmTransferPnPLeftAxisY, controlNode := "Unit1.Em5.ControlNodes".cmTransferPnPLeftAxisY, busy =>, actualPosition =>, actualSpeed =>)
   END_RUNG
   // the same network as SCL:
   #instCmTransferPnPLeftAxisY(enable := TRUE,   // "LBC_Axis64Pos_TecPlcCn"
                           enableManualCmds := #statEnableManualCmds,
                           interlockGeneral := "Unit1.Em5.ControlNodes".cm.interlock.transferPnPLeftAxisY.permit.general,
                           interlockJogForward := "Unit1.Em5.ControlNodes".cm.interlock.transferPnPLeftAxisY.permit.jogForward,
                           interlockJogBackward := "Unit1.Em5.ControlNodes".cm.interlock.transferPnPLeftAxisY.permit.jogBackward,
                           moduleAccessPoint := "BA060AZSICU3~BA060AZSICU3_X150~BA060AZSIDR13_ModuleAccessP,,,",
                           axisNo := 16#5,
                           axis := "BA060AZSIDR13_TransferPnPLeftAxisY",
                           configuration := "Unit1.Em5.Config".cmTransferPnPLeftAxisY,
                           moduleInterface := "Unit1.Em5.HmiInterface".cmTransferPnPLeftAxisY,
                           controlNode := "Unit1.Em5.ControlNodes".cmTransferPnPLeftAxisY);
END_REGION

REGION Network 124: Transfer PnP Left AxisY Softcam
   RUNG wire#powerrail
      "LER_SoftCam_Interface_FC"(actualPosition := "Unit1.Em5.ControlNodes".cmTransferPnPLeftAxisY.monitoring.actualPosition, selectSetPosition := "Unit1.Em5.HmiInterface".cmTransferPnPLeftAxisY.monitoring.selectSetPosition, softCam := "Unit1.Em5.Config".softcam.TransferPnPLeftAxisY, position := "Unit1.Em5.Config".cmTransferPnPLeftAxisY.setPositions, range := 1.0, softCamPos => "Unit1.Em5.ControlNodes".cm.softcam.transferPnPLeftAxisY)
   END_RUNG
   // the same network as SCL:
   "LER_SoftCam_Interface_FC"(actualPosition := "Unit1.Em5.ControlNodes".cmTransferPnPLeftAxisY.monitoring.actualPosition,
                           selectSetPosition := "Unit1.Em5.HmiInterface".cmTransferPnPLeftAxisY.monitoring.selectSetPosition,
                           softCam := "Unit1.Em5.Config".softcam.TransferPnPLeftAxisY,
                           position := "Unit1.Em5.Config".cmTransferPnPLeftAxisY.setPositions,
                           range := 1.0,
                           softCamPos => "Unit1.Em5.ControlNodes".cm.softcam.transferPnPLeftAxisY);
END_REGION

REGION Network 126: Transfer P&P Left Z-Axis Upload Actual Current And Torque Values
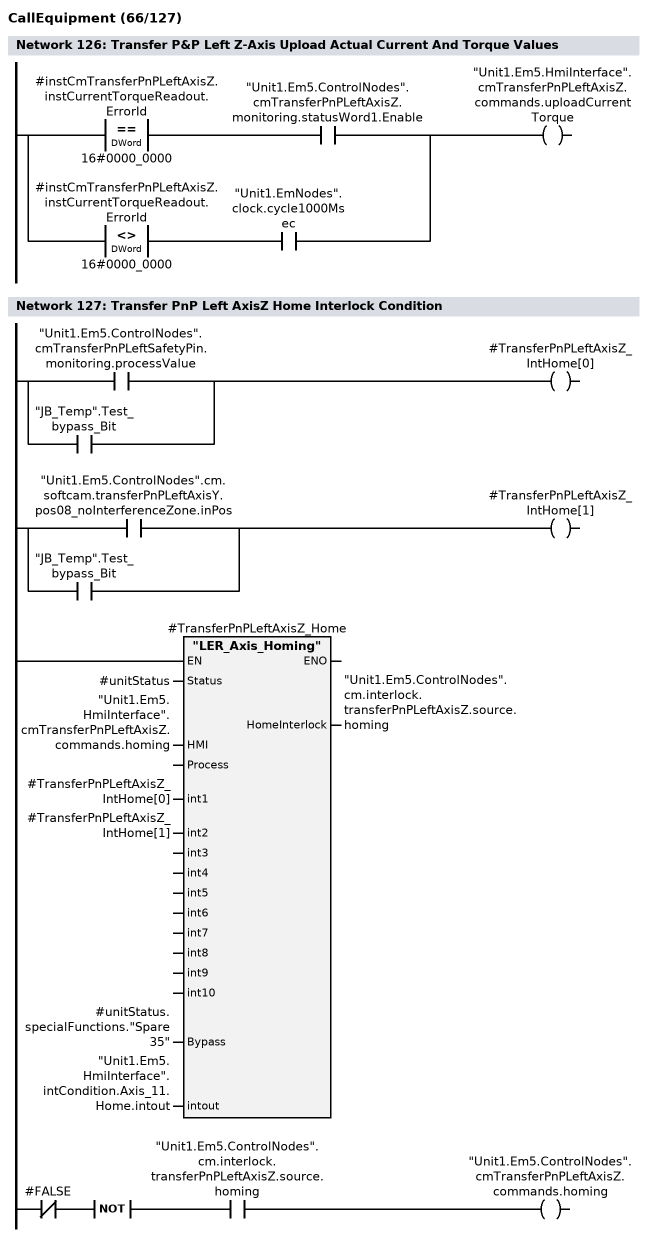
   RUNG wire#powerrail
      { S7_Templates := "SrcType := DWord" } EQ_Contact(in1 := #instCmTransferPnPLeftAxisZ.instCurrentTorqueReadout.ErrorId, in2 := 16#0000_0000)
      Contact( "Unit1.Em5.ControlNodes".cmTransferPnPLeftAxisZ.monitoring.statusWord1.Enable )
      wire#w1
      Coil( "Unit1.Em5.HmiInterface".cmTransferPnPLeftAxisZ.commands.uploadCurrentTorque )
   END_RUNG
   RUNG wire#powerrail
      { S7_Templates := "SrcType := DWord" } NE_Contact(in1 := #instCmTransferPnPLeftAxisZ.instCurrentTorqueReadout.ErrorId, in2 := 16#0000_0000)
      Contact( "Unit1.EmNodes".clock.cycle1000Msec )
   END_RUNG wire#w1
   // the same network as SCL:
   "Unit1.Em5.HmiInterface".cmTransferPnPLeftAxisZ.commands.uploadCurrentTorque := ((#instCmTransferPnPLeftAxisZ.instCurrentTorqueReadout.ErrorId = 16#0000_0000) AND "Unit1.Em5.ControlNodes".cmTransferPnPLeftAxisZ.monitoring.statusWord1.Enable) OR ((#instCmTransferPnPLeftAxisZ.instCurrentTorqueReadout.ErrorId <> 16#0000_0000) AND "Unit1.EmNodes".clock.cycle1000Msec);
END_REGION

REGION Network 127: Transfer PnP Left AxisZ Home Interlock Condition
   RUNG wire#powerrail
      Contact( "Unit1.Em5.ControlNodes".cmTransferPnPLeftSafetyPin.monitoring.processValue )
      wire#w1
      Coil( #TransferPnPLeftAxisZ_IntHome[0] )
   END_RUNG
   RUNG wire#powerrail
      Contact( "JB_Temp".Test_bypass_Bit )
   END_RUNG wire#w1
   RUNG wire#powerrail
      Contact( "Unit1.Em5.ControlNodes".cm.softcam.transferPnPLeftAxisY.pos08_noInterferenceZone.inPos )
      wire#w2
      Coil( #TransferPnPLeftAxisZ_IntHome[1] )
   END_RUNG
   RUNG wire#powerrail
      Contact( "JB_Temp".Test_bypass_Bit )
   END_RUNG wire#w2
   RUNG wire#powerrail
      #TransferPnPLeftAxisZ_Home(Status := #unitStatus, HMI := "Unit1.Em5.HmiInterface".cmTransferPnPLeftAxisZ.commands.homing, Process :=, int1 := #TransferPnPLeftAxisZ_IntHome[0], int2 := #TransferPnPLeftAxisZ_IntHome[1], int3 :=, int4 :=, int5 :=, int6 :=, int7 :=, int8 :=, int9 :=, int10 :=, Bypass := #unitStatus.specialFunctions."Spare 35", intout := "Unit1.Em5.HmiInterface".intCondition.Axis_11.Home.intout, HomeInterlock => "Unit1.Em5.ControlNodes".cm.interlock.transferPnPLeftAxisZ.source.homing)
   END_RUNG
   RUNG wire#powerrail
      I_Contact( #FALSE )
      Not()
      Contact( "Unit1.Em5.ControlNodes".cm.interlock.transferPnPLeftAxisZ.source.homing )
      Coil( "Unit1.Em5.ControlNodes".cmTransferPnPLeftAxisZ.commands.homing )
   END_RUNG
   // the same network as SCL:
   #TransferPnPLeftAxisZ_IntHome[0] := "Unit1.Em5.ControlNodes".cmTransferPnPLeftSafetyPin.monitoring.processValue OR "JB_Temp".Test_bypass_Bit;
   #TransferPnPLeftAxisZ_IntHome[1] := "Unit1.Em5.ControlNodes".cm.softcam.transferPnPLeftAxisY.pos08_noInterferenceZone.inPos OR "JB_Temp".Test_bypass_Bit;
   #TransferPnPLeftAxisZ_Home(Status := #unitStatus,   // "LER_Axis_Homing"
                           HMI := "Unit1.Em5.HmiInterface".cmTransferPnPLeftAxisZ.commands.homing,
                           int1 := #TransferPnPLeftAxisZ_IntHome[0],
                           int2 := #TransferPnPLeftAxisZ_IntHome[1],
                           Bypass := #unitStatus.specialFunctions."Spare 35",
                           intout := "Unit1.Em5.HmiInterface".intCondition.Axis_11.Home.intout,
                           HomeInterlock => "Unit1.Em5.ControlNodes".cm.interlock.transferPnPLeftAxisZ.source.homing);
   "Unit1.Em5.ControlNodes".cmTransferPnPLeftAxisZ.commands.homing := NOT (NOT #FALSE) AND "Unit1.Em5.ControlNodes".cm.interlock.transferPnPLeftAxisZ.source.homing;
END_REGION

REGION Network 128: Transfer PnP Left AxisZ JOG Interlock Condition
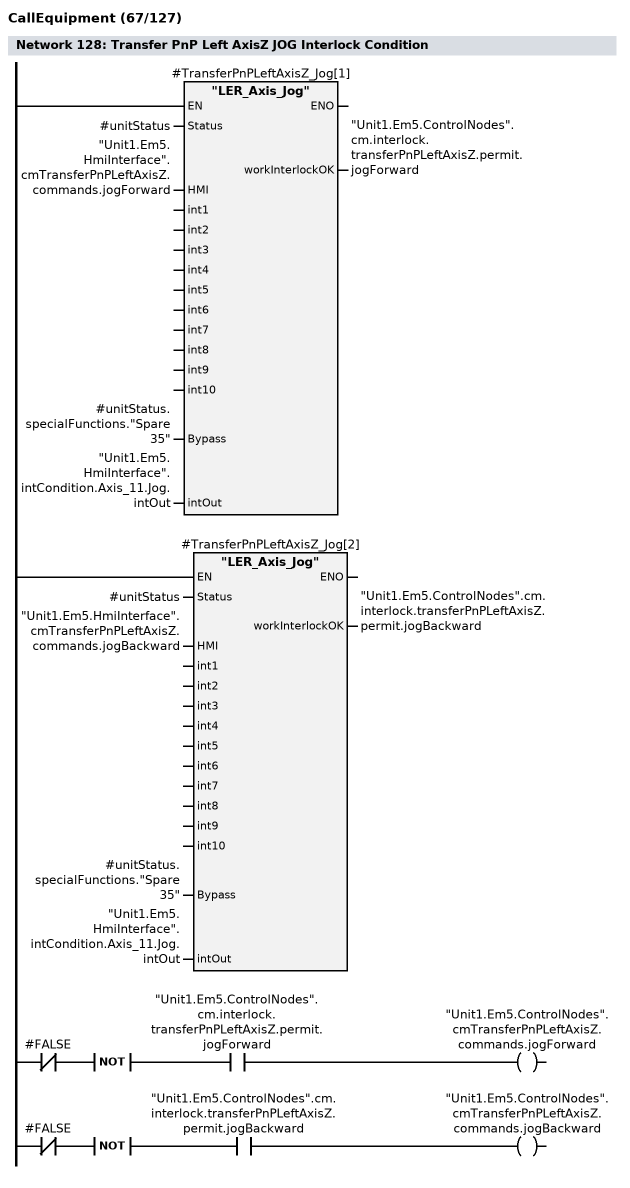
   RUNG wire#powerrail
      #TransferPnPLeftAxisZ_Jog[1](Status := #unitStatus, HMI := "Unit1.Em5.HmiInterface".cmTransferPnPLeftAxisZ.commands.jogForward, int1 :=, int2 :=, int3 :=, int4 :=, int5 :=, int6 :=, int7 :=, int8 :=, int9 :=, int10 :=, Bypass := #unitStatus.specialFunctions."Spare 35", intOut := "Unit1.Em5.HmiInterface".intCondition.Axis_11.Jog.intOut, workInterlockOK => "Unit1.Em5.ControlNodes".cm.interlock.transferPnPLeftAxisZ.permit.jogForward)
   END_RUNG
   RUNG wire#powerrail
      #TransferPnPLeftAxisZ_Jog[2](Status := #unitStatus, HMI := "Unit1.Em5.HmiInterface".cmTransferPnPLeftAxisZ.commands.jogBackward, int1 :=, int2 :=, int3 :=, int4 :=, int5 :=, int6 :=, int7 :=, int8 :=, int9 :=, int10 :=, Bypass := #unitStatus.specialFunctions."Spare 35", intOut := "Unit1.Em5.HmiInterface".intCondition.Axis_11.Jog.intOut, workInterlockOK => "Unit1.Em5.ControlNodes".cm.interlock.transferPnPLeftAxisZ.permit.jogBackward)
   END_RUNG
   RUNG wire#powerrail
      I_Contact( #FALSE )
      Not()
      Contact( "Unit1.Em5.ControlNodes".cm.interlock.transferPnPLeftAxisZ.permit.jogForward )
      Coil( "Unit1.Em5.ControlNodes".cmTransferPnPLeftAxisZ.commands.jogForward )
   END_RUNG
   RUNG wire#powerrail
      I_Contact( #FALSE )
      Not()
      Contact( "Unit1.Em5.ControlNodes".cm.interlock.transferPnPLeftAxisZ.permit.jogBackward )
      Coil( "Unit1.Em5.ControlNodes".cmTransferPnPLeftAxisZ.commands.jogBackward )
   END_RUNG
   // the same network as SCL:
   #TransferPnPLeftAxisZ_Jog[1](Status := #unitStatus,   // "LER_Axis_Jog"
                           HMI := "Unit1.Em5.HmiInterface".cmTransferPnPLeftAxisZ.commands.jogForward,
                           Bypass := #unitStatus.specialFunctions."Spare 35",
                           intOut := "Unit1.Em5.HmiInterface".intCondition.Axis_11.Jog.intOut,
                           workInterlockOK => "Unit1.Em5.ControlNodes".cm.interlock.transferPnPLeftAxisZ.permit.jogForward);
   #TransferPnPLeftAxisZ_Jog[2](Status := #unitStatus,   // "LER_Axis_Jog"
                           HMI := "Unit1.Em5.HmiInterface".cmTransferPnPLeftAxisZ.commands.jogBackward,
                           Bypass := #unitStatus.specialFunctions."Spare 35",
                           intOut := "Unit1.Em5.HmiInterface".intCondition.Axis_11.Jog.intOut,
                           workInterlockOK => "Unit1.Em5.ControlNodes".cm.interlock.transferPnPLeftAxisZ.permit.jogBackward);
   "Unit1.Em5.ControlNodes".cmTransferPnPLeftAxisZ.commands.jogForward := NOT (NOT #FALSE) AND "Unit1.Em5.ControlNodes".cm.interlock.transferPnPLeftAxisZ.permit.jogForward;
   "Unit1.Em5.ControlNodes".cmTransferPnPLeftAxisZ.commands.jogBackward := NOT (NOT #FALSE) AND "Unit1.Em5.ControlNodes".cm.interlock.transferPnPLeftAxisZ.permit.jogBackward;
END_REGION

REGION Network 129: Transfer PnP Left AxisZ Position Absolute Position0
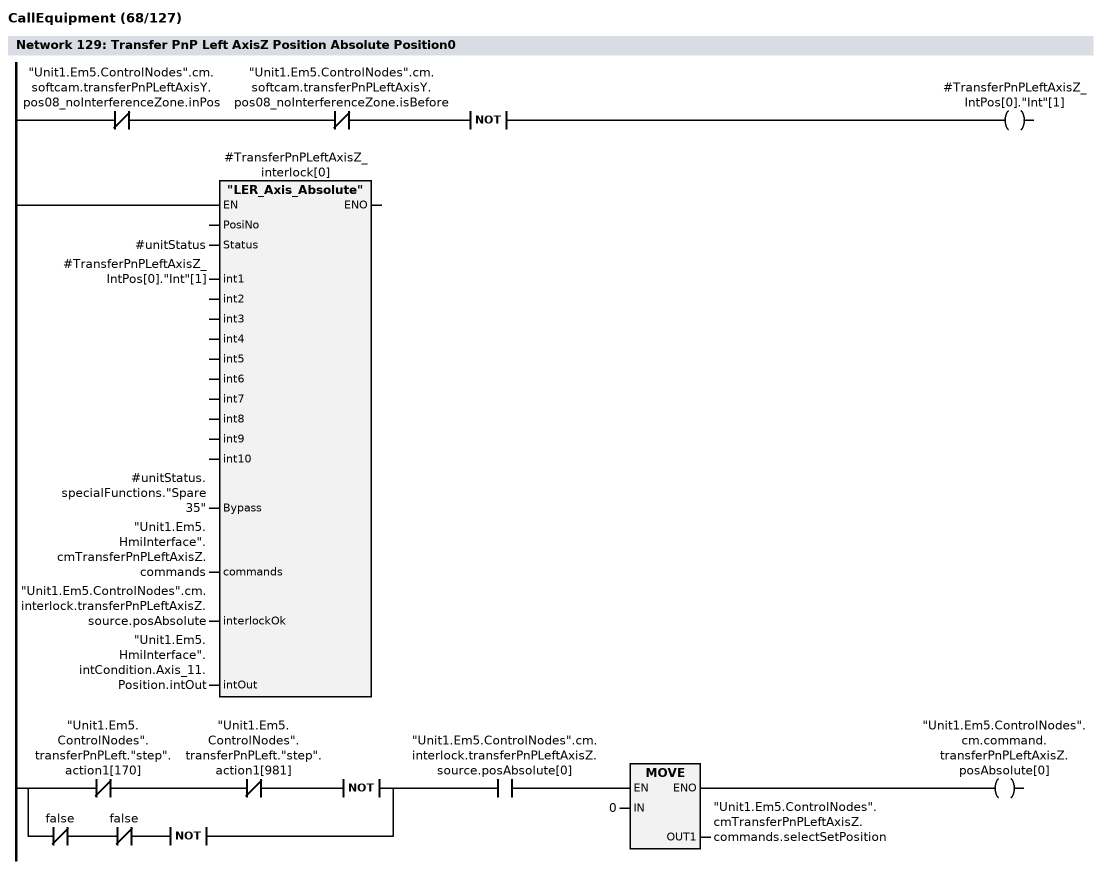
   RUNG wire#powerrail
      I_Contact( "Unit1.Em5.ControlNodes".cm.softcam.transferPnPLeftAxisY.pos08_noInterferenceZone.inPos )
      I_Contact( "Unit1.Em5.ControlNodes".cm.softcam.transferPnPLeftAxisY.pos08_noInterferenceZone.isBefore )
      Not()
      Coil( #TransferPnPLeftAxisZ_IntPos[0]."Int"[1] )
   END_RUNG
   RUNG wire#powerrail
      #TransferPnPLeftAxisZ_interlock[0](PosiNo :=, Status := #unitStatus, int1 := #TransferPnPLeftAxisZ_IntPos[0]."Int"[1], int2 :=, int3 :=, int4 :=, int5 :=, int6 :=, int7 :=, int8 :=, int9 :=, int10 :=, Bypass := #unitStatus.specialFunctions."Spare 35", commands := "Unit1.Em5.HmiInterface".cmTransferPnPLeftAxisZ.commands, interlockOk := "Unit1.Em5.ControlNodes".cm.interlock.transferPnPLeftAxisZ.source.posAbsolute, intOut := "Unit1.Em5.HmiInterface".intCondition.Axis_11.Position.intOut)
   END_RUNG
   RUNG wire#powerrail
      I_Contact( "Unit1.Em5.ControlNodes".transferPnPLeft."step".action1[170] )
      I_Contact( "Unit1.Em5.ControlNodes".transferPnPLeft."step".action1[981] )
      Not()
      wire#w1
      Contact( "Unit1.Em5.ControlNodes".cm.interlock.transferPnPLeftAxisZ.source.posAbsolute[0] )
      Move(in := 0, out1 => "Unit1.Em5.ControlNodes".cmTransferPnPLeftAxisZ.commands.selectSetPosition)
      Coil( "Unit1.Em5.ControlNodes".cm.command.transferPnPLeftAxisZ.posAbsolute[0] )
   END_RUNG
   RUNG wire#powerrail
      I_Contact( false )
      I_Contact( false )
      Not()
   END_RUNG wire#w1
   // the same network as SCL:
   #TransferPnPLeftAxisZ_IntPos[0]."Int"[1] := NOT (NOT "Unit1.Em5.ControlNodes".cm.softcam.transferPnPLeftAxisY.pos08_noInterferenceZone.inPos AND NOT "Unit1.Em5.ControlNodes".cm.softcam.transferPnPLeftAxisY.pos08_noInterferenceZone.isBefore);
   #TransferPnPLeftAxisZ_interlock[0](Status := #unitStatus,   // "LER_Axis_Absolute"
                           int1 := #TransferPnPLeftAxisZ_IntPos[0]."Int"[1],
                           Bypass := #unitStatus.specialFunctions."Spare 35",
                           commands := "Unit1.Em5.HmiInterface".cmTransferPnPLeftAxisZ.commands,
                           interlockOk := "Unit1.Em5.ControlNodes".cm.interlock.transferPnPLeftAxisZ.source.posAbsolute,
                           intOut := "Unit1.Em5.HmiInterface".intCondition.Axis_11.Position.intOut);
   #_w1 := (NOT (NOT "Unit1.Em5.ControlNodes".transferPnPLeft."step".action1[170] AND NOT "Unit1.Em5.ControlNodes".transferPnPLeft."step".action1[981]) OR NOT (NOT false AND NOT false)) AND "Unit1.Em5.ControlNodes".cm.interlock.transferPnPLeftAxisZ.source.posAbsolute[0];
   IF #_w1 THEN "Unit1.Em5.ControlNodes".cmTransferPnPLeftAxisZ.commands.selectSetPosition := 0; END_IF;
   "Unit1.Em5.ControlNodes".cm.command.transferPnPLeftAxisZ.posAbsolute[0] := #_w1;
END_REGION

REGION Network 130: Transfer PnP Left AxisZ Position Absolute Position1
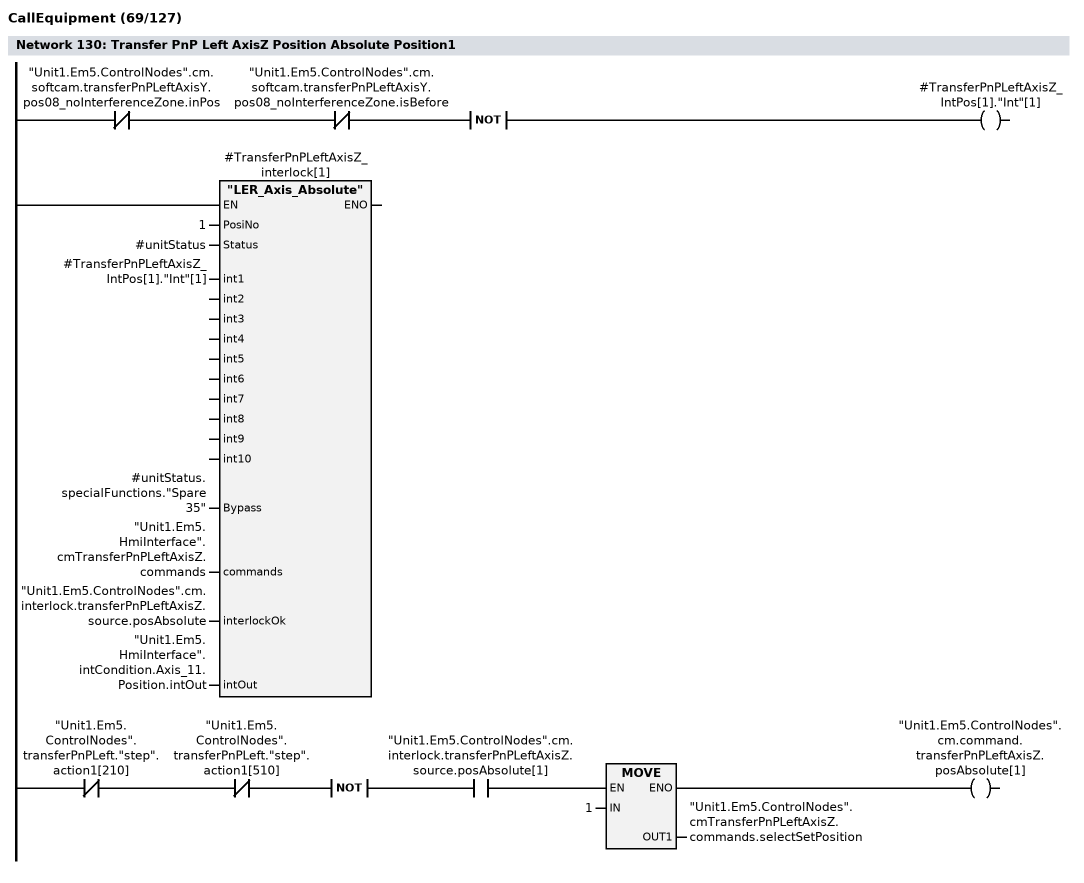
   RUNG wire#powerrail
      I_Contact( "Unit1.Em5.ControlNodes".cm.softcam.transferPnPLeftAxisY.pos08_noInterferenceZone.inPos )
      I_Contact( "Unit1.Em5.ControlNodes".cm.softcam.transferPnPLeftAxisY.pos08_noInterferenceZone.isBefore )
      Not()
      Coil( #TransferPnPLeftAxisZ_IntPos[1]."Int"[1] )
   END_RUNG
   RUNG wire#powerrail
      #TransferPnPLeftAxisZ_interlock[1](PosiNo := 1, Status := #unitStatus, int1 := #TransferPnPLeftAxisZ_IntPos[1]."Int"[1], int2 :=, int3 :=, int4 :=, int5 :=, int6 :=, int7 :=, int8 :=, int9 :=, int10 :=, Bypass := #unitStatus.specialFunctions."Spare 35", commands := "Unit1.Em5.HmiInterface".cmTransferPnPLeftAxisZ.commands, interlockOk := "Unit1.Em5.ControlNodes".cm.interlock.transferPnPLeftAxisZ.source.posAbsolute, intOut := "Unit1.Em5.HmiInterface".intCondition.Axis_11.Position.intOut)
   END_RUNG
   RUNG wire#powerrail
      I_Contact( "Unit1.Em5.ControlNodes".transferPnPLeft."step".action1[210] )
      I_Contact( "Unit1.Em5.ControlNodes".transferPnPLeft."step".action1[510] )
      Not()
      Contact( "Unit1.Em5.ControlNodes".cm.interlock.transferPnPLeftAxisZ.source.posAbsolute[1] )
      Move(in := 1, out1 => "Unit1.Em5.ControlNodes".cmTransferPnPLeftAxisZ.commands.selectSetPosition)
      Coil( "Unit1.Em5.ControlNodes".cm.command.transferPnPLeftAxisZ.posAbsolute[1] )
   END_RUNG
   // the same network as SCL:
   #TransferPnPLeftAxisZ_IntPos[1]."Int"[1] := NOT (NOT "Unit1.Em5.ControlNodes".cm.softcam.transferPnPLeftAxisY.pos08_noInterferenceZone.inPos AND NOT "Unit1.Em5.ControlNodes".cm.softcam.transferPnPLeftAxisY.pos08_noInterferenceZone.isBefore);
   #TransferPnPLeftAxisZ_interlock[1](PosiNo := 1,   // "LER_Axis_Absolute"
                           Status := #unitStatus,
                           int1 := #TransferPnPLeftAxisZ_IntPos[1]."Int"[1],
                           Bypass := #unitStatus.specialFunctions."Spare 35",
                           commands := "Unit1.Em5.HmiInterface".cmTransferPnPLeftAxisZ.commands,
                           interlockOk := "Unit1.Em5.ControlNodes".cm.interlock.transferPnPLeftAxisZ.source.posAbsolute,
                           intOut := "Unit1.Em5.HmiInterface".intCondition.Axis_11.Position.intOut);
   #_w1 := NOT (NOT "Unit1.Em5.ControlNodes".transferPnPLeft."step".action1[210] AND NOT "Unit1.Em5.ControlNodes".transferPnPLeft."step".action1[510]) AND "Unit1.Em5.ControlNodes".cm.interlock.transferPnPLeftAxisZ.source.posAbsolute[1];
   IF #_w1 THEN "Unit1.Em5.ControlNodes".cmTransferPnPLeftAxisZ.commands.selectSetPosition := 1; END_IF;
   "Unit1.Em5.ControlNodes".cm.command.transferPnPLeftAxisZ.posAbsolute[1] := #_w1;
END_REGION

REGION Network 131: Transfer PnP Left AxisZ Position Absolute Position2
